    fTable_Be[559, 0] := 2194.37; fTable_Be[559, 1] := 4.04346; fTable_Be[559, 2] := 0.0262870;
    fTable_Be[560, 0] := 2229.86; fTable_Be[560, 1] := 4.04236; fTable_Be[560, 2] := 0.0254127;
    fTable_Be[561, 0] := 2265.93; fTable_Be[561, 1] := 4.04127; fTable_Be[561, 2] := 0.0245675;
    fTable_Be[562, 0] := 2302.57; fTable_Be[562, 1] := 4.04021; fTable_Be[562, 2] := 0.0237503;
    fTable_Be[563, 0] := 2339.82; fTable_Be[563, 1] := 4.03918; fTable_Be[563, 2] := 0.0229604;
    fTable_Be[564, 0] := 2377.66; fTable_Be[564, 1] := 4.03817; fTable_Be[564, 2] := 0.0221967;
    fTable_Be[565, 0] := 2416.12; fTable_Be[565, 1] := 4.03718; fTable_Be[565, 2] := 0.0214584;
    fTable_Be[566, 0] := 2455.20; fTable_Be[566, 1] := 4.03621; fTable_Be[566, 2] := 0.0207447;
    fTable_Be[567, 0] := 2494.91; fTable_Be[567, 1] := 4.03527; fTable_Be[567, 2] := 0.0200547;
    fTable_Be[568, 0] := 2535.26; fTable_Be[568, 1] := 4.03435; fTable_Be[568, 2] := 0.0193877;
    fTable_Be[569, 0] := 2576.27; fTable_Be[569, 1] := 4.03345; fTable_Be[569, 2] := 0.0187429;
    fTable_Be[570, 0] := 2617.94; fTable_Be[570, 1] := 4.03257; fTable_Be[570, 2] := 0.0181195;
    fTable_Be[571, 0] := 2660.28; fTable_Be[571, 1] := 4.03171; fTable_Be[571, 2] := 0.0175168;
    fTable_Be[572, 0] := 2703.31; fTable_Be[572, 1] := 4.03088; fTable_Be[572, 2] := 0.0169342;
    fTable_Be[573, 0] := 2747.03; fTable_Be[573, 1] := 4.03006; fTable_Be[573, 2] := 0.0163709;
    fTable_Be[574, 0] := 2791.46; fTable_Be[574, 1] := 4.02926; fTable_Be[574, 2] := 0.0158264;
    fTable_Be[575, 0] := 2836.61; fTable_Be[575, 1] := 4.02849; fTable_Be[575, 2] := 0.0153000;
    fTable_Be[576, 0] := 2882.49; fTable_Be[576, 1] := 4.02773; fTable_Be[576, 2] := 0.0147911;
    fTable_Be[577, 0] := 2929.11; fTable_Be[577, 1] := 4.02700; fTable_Be[577, 2] := 0.0142992;
    fTable_Be[578, 0] := 2976.49; fTable_Be[578, 1] := 4.02628; fTable_Be[578, 2] := 0.0138236;
    fTable_Be[579, 0] := 3024.63; fTable_Be[579, 1] := 4.02559; fTable_Be[579, 2] := 0.0133638;
    fTable_Be[580, 0] := 3073.55; fTable_Be[580, 1] := 4.02491; fTable_Be[580, 2] := 0.0129072;
    fTable_Be[581, 0] := 3123.26; fTable_Be[581, 1] := 4.02424; fTable_Be[581, 2] := 0.0124663;
    fTable_Be[582, 0] := 3173.78; fTable_Be[582, 1] := 4.02359; fTable_Be[582, 2] := 0.0120403;
    fTable_Be[583, 0] := 3225.11; fTable_Be[583, 1] := 4.02295; fTable_Be[583, 2] := 0.0116290;
    fTable_Be[584, 0] := 3277.28; fTable_Be[584, 1] := 4.02233; fTable_Be[584, 2] := 0.0112317;
    fTable_Be[585, 0] := 3330.29; fTable_Be[585, 1] := 4.02172; fTable_Be[585, 2] := 0.0108480;
    fTable_Be[586, 0] := 3384.15; fTable_Be[586, 1] := 4.02113; fTable_Be[586, 2] := 0.0104774;
    fTable_Be[587, 0] := 3438.89; fTable_Be[587, 1] := 4.02055; fTable_Be[587, 2] := 0.0101194;
    fTable_Be[588, 0] := 3494.51; fTable_Be[588, 1] := 4.01998; fTable_Be[588, 2] := 0.00977365;
    fTable_Be[589, 0] := 3551.03; fTable_Be[589, 1] := 4.01943; fTable_Be[589, 2] := 0.00943974;
    fTable_Be[590, 0] := 3608.46; fTable_Be[590, 1] := 4.01890; fTable_Be[590, 2] := 0.00911724;
    fTable_Be[591, 0] := 3666.83; fTable_Be[591, 1] := 4.01837; fTable_Be[591, 2] := 0.00880575;
    fTable_Be[592, 0] := 3726.13; fTable_Be[592, 1] := 4.01786; fTable_Be[592, 2] := 0.00850491;
    fTable_Be[593, 0] := 3786.40; fTable_Be[593, 1] := 4.01736; fTable_Be[593, 2] := 0.00821432;
    fTable_Be[594, 0] := 3847.64; fTable_Be[594, 1] := 4.01688; fTable_Be[594, 2] := 0.00793369;
    fTable_Be[595, 0] := 3909.88; fTable_Be[595, 1] := 4.01641; fTable_Be[595, 2] := 0.00766264;
    fTable_Be[596, 0] := 3973.12; fTable_Be[596, 1] := 4.01595; fTable_Be[596, 2] := 0.00740085;
    fTable_Be[597, 0] := 4037.38; fTable_Be[597, 1] := 4.01550; fTable_Be[597, 2] := 0.00714801;
    fTable_Be[598, 0] := 4102.68; fTable_Be[598, 1] := 4.01506; fTable_Be[598, 2] := 0.00690380;
    fTable_Be[599, 0] := 4169.04; fTable_Be[599, 1] := 4.01464; fTable_Be[599, 2] := 0.00666401;
    fTable_Be[600, 0] := 4236.47; fTable_Be[600, 1] := 4.01423; fTable_Be[600, 2] := 0.00643256;
    fTable_Be[601, 0] := 4304.99; fTable_Be[601, 1] := 4.01382; fTable_Be[601, 2] := 0.00620915;
    fTable_Be[602, 0] := 4374.62; fTable_Be[602, 1] := 4.01343; fTable_Be[602, 2] := 0.00599350;
    fTable_Be[603, 0] := 4445.37; fTable_Be[603, 1] := 4.01304; fTable_Be[603, 2] := 0.00578535;
    fTable_Be[604, 0] := 4517.27; fTable_Be[604, 1] := 4.01267; fTable_Be[604, 2] := 0.00558442;
    fTable_Be[605, 0] := 4590.34; fTable_Be[605, 1] := 4.01230; fTable_Be[605, 2] := 0.00539045;
    fTable_Be[606, 0] := 4664.58; fTable_Be[606, 1] := 4.01195; fTable_Be[606, 2] := 0.00520323;
    fTable_Be[607, 0] := 4740.03; fTable_Be[607, 1] := 4.01160; fTable_Be[607, 2] := 0.00502252;
    fTable_Be[608, 0] := 4816.70; fTable_Be[608, 1] := 4.01126; fTable_Be[608, 2] := 0.00484809;
    fTable_Be[609, 0] := 4894.60; fTable_Be[609, 1] := 4.01093; fTable_Be[609, 2] := 0.00467971;
    fTable_Be[610, 0] := 4973.77; fTable_Be[610, 1] := 4.01061; fTable_Be[610, 2] := 0.00451716;
    fTable_Be[611, 0] := 5054.21; fTable_Be[611, 1] := 4.01030; fTable_Be[611, 2] := 0.00436028;
    fTable_Be[612, 0] := 5135.96; fTable_Be[612, 1] := 4.01000; fTable_Be[612, 2] := 0.00420884;
    fTable_Be[613, 0] := 5219.03; fTable_Be[613, 1] := 4.00970; fTable_Be[613, 2] := 0.00406267;
    fTable_Be[614, 0] := 5303.45; fTable_Be[614, 1] := 4.00941; fTable_Be[614, 2] := 0.00391977;
    fTable_Be[615, 0] := 5389.23; fTable_Be[615, 1] := 4.00913; fTable_Be[615, 2] := 0.00378191;
    fTable_Be[616, 0] := 5476.39; fTable_Be[616, 1] := 4.00886; fTable_Be[616, 2] := 0.00364888;
    fTable_Be[617, 0] := 5564.97; fTable_Be[617, 1] := 4.00860; fTable_Be[617, 2] := 0.00352054;
    fTable_Be[618, 0] := 5654.98; fTable_Be[618, 1] := 4.00834; fTable_Be[618, 2] := 0.00339671;
    fTable_Be[619, 0] := 5746.44; fTable_Be[619, 1] := 4.00808; fTable_Be[619, 2] := 0.00327724;
    fTable_Be[620, 0] := 5839.39; fTable_Be[620, 1] := 4.00784; fTable_Be[620, 2] := 0.00316197;
    fTable_Be[621, 0] := 5933.83; fTable_Be[621, 1] := 4.00760; fTable_Be[621, 2] := 0.00305075;
    fTable_Be[622, 0] := 6029.81; fTable_Be[622, 1] := 4.00737; fTable_Be[622, 2] := 0.00294344;
    fTable_Be[623, 0] := 6127.33; fTable_Be[623, 1] := 4.00714; fTable_Be[623, 2] := 0.00283992;
    fTable_Be[624, 0] := 6226.44; fTable_Be[624, 1] := 4.00692; fTable_Be[624, 2] := 0.00274003;
    fTable_Be[625, 0] := 6327.15; fTable_Be[625, 1] := 4.00671; fTable_Be[625, 2] := 0.00264365;
    fTable_Be[626, 0] := 6429.48; fTable_Be[626, 1] := 4.00650; fTable_Be[626, 2] := 0.00254975;
    fTable_Be[627, 0] := 6533.48; fTable_Be[627, 1] := 4.00630; fTable_Be[627, 2] := 0.00245918;
    fTable_Be[628, 0] := 6639.15; fTable_Be[628, 1] := 4.00610; fTable_Be[628, 2] := 0.00237183;
    fTable_Be[629, 0] := 6746.53; fTable_Be[629, 1] := 4.00591; fTable_Be[629, 2] := 0.00228759;
    fTable_Be[630, 0] := 6855.65; fTable_Be[630, 1] := 4.00572; fTable_Be[630, 2] := 0.00220633;
    fTable_Be[631, 0] := 6966.54; fTable_Be[631, 1] := 4.00554; fTable_Be[631, 2] := 0.00212796;
    fTable_Be[632, 0] := 7079.21; fTable_Be[632, 1] := 4.00536; fTable_Be[632, 2] := 0.00205238;
    fTable_Be[633, 0] := 7193.71; fTable_Be[633, 1] := 4.00519; fTable_Be[633, 2] := 0.00197947;
    fTable_Be[634, 0] := 7310.07; fTable_Be[634, 1] := 4.00502; fTable_Be[634, 2] := 0.00190916;
    fTable_Be[635, 0] := 7428.30; fTable_Be[635, 1] := 4.00485; fTable_Be[635, 2] := 0.00184135;
    fTable_Be[636, 0] := 7548.45; fTable_Be[636, 1] := 4.00469; fTable_Be[636, 2] := 0.00177595;
    fTable_Be[637, 0] := 7670.54; fTable_Be[637, 1] := 4.00454; fTable_Be[637, 2] := 0.00171287;
    fTable_Be[638, 0] := 7794.60; fTable_Be[638, 1] := 4.00439; fTable_Be[638, 2] := 0.00165202;
    fTable_Be[639, 0] := 7920.68; fTable_Be[639, 1] := 4.00424; fTable_Be[639, 2] := 0.00159334;
    fTable_Be[640, 0] := 8048.79; fTable_Be[640, 1] := 4.00410; fTable_Be[640, 2] := 0.00153675;
    fTable_Be[641, 0] := 8178.97; fTable_Be[641, 1] := 4.00396; fTable_Be[641, 2] := 0.00148216;
    fTable_Be[642, 0] := 8311.26; fTable_Be[642, 1] := 4.00383; fTable_Be[642, 2] := 0.00142952;
    fTable_Be[643, 0] := 8445.68; fTable_Be[643, 1] := 4.00370; fTable_Be[643, 2] := 0.00137819;
    fTable_Be[644, 0] := 8582.29; fTable_Be[644, 1] := 4.00357; fTable_Be[644, 2] := 0.00132870;
    fTable_Be[645, 0] := 8721.10; fTable_Be[645, 1] := 4.00345; fTable_Be[645, 2] := 0.00128099;
    fTable_Be[646, 0] := 8862.16; fTable_Be[646, 1] := 4.00333; fTable_Be[646, 2] := 0.00123499;
    fTable_Be[647, 0] := 9005.49; fTable_Be[647, 1] := 4.00321; fTable_Be[647, 2] := 0.00119064;
    fTable_Be[648, 0] := 9151.15; fTable_Be[648, 1] := 4.00310; fTable_Be[648, 2] := 0.00114789;
    fTable_Be[649, 0] := 9299.16; fTable_Be[649, 1] := 4.00299; fTable_Be[649, 2] := 0.00110667;
    fTable_Be[650, 0] := 9449.57; fTable_Be[650, 1] := 4.00288; fTable_Be[650, 2] := 0.00106693;
    fTable_Be[651, 0] := 9602.41; fTable_Be[651, 1] := 4.00277; fTable_Be[651, 2] := 0.00102862;
    fTable_Be[652, 0] := 9757.72; fTable_Be[652, 1] := 4.00267; fTable_Be[652, 2] := 0.000991686;
    fTable_Be[653, 0] := 9915.54; fTable_Be[653, 1] := 4.00257; fTable_Be[653, 2] := 0.000956077;
    fTable_Be[654, 0] := 10075.9; fTable_Be[654, 1] := 4.00248; fTable_Be[654, 2] := 0.000921746;
    fTable_Be[655, 0] := 10238.9; fTable_Be[655, 1] := 4.00238; fTable_Be[655, 2] := 0.000888646;
    fTable_Be[656, 0] := 10404.5; fTable_Be[656, 1] := 4.00229; fTable_Be[656, 2] := 0.000856737;
    fTable_Be[657, 0] := 10572.8; fTable_Be[657, 1] := 4.00221; fTable_Be[657, 2] := 0.000825973;
    fTable_Be[658, 0] := 10743.8; fTable_Be[658, 1] := 4.00212; fTable_Be[658, 2] := 0.000796314;
    fTable_Be[659, 0] := 10917.6; fTable_Be[659, 1] := 4.00204; fTable_Be[659, 2] := 0.000767721;
    fTable_Be[660, 0] := 11094.1; fTable_Be[660, 1] := 4.00196; fTable_Be[660, 2] := 0.000740154;
    fTable_Be[661, 0] := 11273.6; fTable_Be[661, 1] := 4.00188; fTable_Be[661, 2] := 0.000713574;
    fTable_Be[662, 0] := 11455.9; fTable_Be[662, 1] := 4.00180; fTable_Be[662, 2] := 0.000687952;
    fTable_Be[663, 0] := 11641.2; fTable_Be[663, 1] := 4.00173; fTable_Be[663, 2] := 0.000663249;
    fTable_Be[664, 0] := 11829.5; fTable_Be[664, 1] := 4.00165; fTable_Be[664, 2] := 0.000639433;
    fTable_Be[665, 0] := 12020.8; fTable_Be[665, 1] := 4.00158; fTable_Be[665, 2] := 0.000616473;
    fTable_Be[666, 0] := 12215.3; fTable_Be[666, 1] := 4.00152; fTable_Be[666, 2] := 0.000594337;
    fTable_Be[667, 0] := 12412.8; fTable_Be[667, 1] := 4.00145; fTable_Be[667, 2] := 0.000572994;
    fTable_Be[668, 0] := 12613.6; fTable_Be[668, 1] := 4.00139; fTable_Be[668, 2] := 0.000552174;
    fTable_Be[669, 0] := 12817.6; fTable_Be[669, 1] := 4.00132; fTable_Be[669, 2] := 0.000532111;
    fTable_Be[670, 0] := 13024.9; fTable_Be[670, 1] := 4.00126; fTable_Be[670, 2] := 0.000512776;
    fTable_Be[671, 0] := 13235.6; fTable_Be[671, 1] := 4.00120; fTable_Be[671, 2] := 0.000494145;
    fTable_Be[672, 0] := 13449.7; fTable_Be[672, 1] := 4.00115; fTable_Be[672, 2] := 0.000476188;
    fTable_Be[673, 0] := 13667.2; fTable_Be[673, 1] := 4.00109; fTable_Be[673, 2] := 0.000458886;
    fTable_Be[674, 0] := 13888.3; fTable_Be[674, 1] := 4.00104; fTable_Be[674, 2] := 0.000442212;
    fTable_Be[675, 0] := 14112.9; fTable_Be[675, 1] := 4.00098; fTable_Be[675, 2] := 0.000426144;
    fTable_Be[676, 0] := 14341.2; fTable_Be[676, 1] := 4.00093; fTable_Be[676, 2] := 0.000410660;
    fTable_Be[677, 0] := 14573.1; fTable_Be[677, 1] := 4.00088; fTable_Be[677, 2] := 0.000395739;
    fTable_Be[678, 0] := 14808.8; fTable_Be[678, 1] := 4.00083; fTable_Be[678, 2] := 0.000381358;
    fTable_Be[679, 0] := 15048.3; fTable_Be[679, 1] := 4.00079; fTable_Be[679, 2] := 0.000367502;
    fTable_Be[680, 0] := 15291.7; fTable_Be[680, 1] := 4.00074; fTable_Be[680, 2] := 0.000354148;
    fTable_Be[681, 0] := 15539.1; fTable_Be[681, 1] := 4.00070; fTable_Be[681, 2] := 0.000341280;
    fTable_Be[682, 0] := 15790.4; fTable_Be[682, 1] := 4.00065; fTable_Be[682, 2] := 0.000328880;
    fTable_Be[683, 0] := 16045.8; fTable_Be[683, 1] := 4.00061; fTable_Be[683, 2] := 0.000316929;
    fTable_Be[684, 0] := 16305.3; fTable_Be[684, 1] := 4.00057; fTable_Be[684, 2] := 0.000305413;
    fTable_Be[685, 0] := 16569.1; fTable_Be[685, 1] := 4.00053; fTable_Be[685, 2] := 0.000294207;
    fTable_Be[686, 0] := 16837.0; fTable_Be[686, 1] := 4.00049; fTable_Be[686, 2] := 0.000283413;
    fTable_Be[687, 0] := 17109.4; fTable_Be[687, 1] := 4.00046; fTable_Be[687, 2] := 0.000273015;
    fTable_Be[688, 0] := 17386.1; fTable_Be[688, 1] := 4.00042; fTable_Be[688, 2] := 0.000262998;
    fTable_Be[689, 0] := 17667.3; fTable_Be[689, 1] := 4.00039; fTable_Be[689, 2] := 0.000253348;
    fTable_Be[690, 0] := 17953.1; fTable_Be[690, 1] := 4.00035; fTable_Be[690, 2] := 0.000244052;
    fTable_Be[691, 0] := 18243.4; fTable_Be[691, 1] := 4.00032; fTable_Be[691, 2] := 0.000235098;
    fTable_Be[692, 0] := 18538.5; fTable_Be[692, 1] := 4.00029; fTable_Be[692, 2] := 0.000226472;
    fTable_Be[693, 0] := 18838.4; fTable_Be[693, 1] := 4.00026; fTable_Be[693, 2] := 0.000218163;
    fTable_Be[694, 0] := 19143.0; fTable_Be[694, 1] := 4.00023; fTable_Be[694, 2] := 0.000210159;
    fTable_Be[695, 0] := 19452.7; fTable_Be[695, 1] := 4.00020; fTable_Be[695, 2] := 0.000202447;
    fTable_Be[696, 0] := 19767.3; fTable_Be[696, 1] := 4.00017; fTable_Be[696, 2] := 0.000195019;
    fTable_Be[697, 0] := 20087.0; fTable_Be[697, 1] := 4.00014; fTable_Be[697, 2] := 0.000187864;
    fTable_Be[698, 0] := 20411.9; fTable_Be[698, 1] := 4.00011; fTable_Be[698, 2] := 0.000180971;
    fTable_Be[699, 0] := 20742.1; fTable_Be[699, 1] := 4.00009; fTable_Be[699, 2] := 0.000174332;
    fTable_Be[700, 0] := 21077.5; fTable_Be[700, 1] := 4.00006; fTable_Be[700, 2] := 0.000167935;
    fTable_Be[701, 0] := 21418.5; fTable_Be[701, 1] := 4.00004; fTable_Be[701, 2] := 0.000161773;
    fTable_Be[702, 0] := 21764.9; fTable_Be[702, 1] := 4.00001; fTable_Be[702, 2] := 0.000155838;
    fTable_Be[703, 0] := 22116.9; fTable_Be[703, 1] := 3.99999; fTable_Be[703, 2] := 0.000150120;
    fTable_Be[704, 0] := 22474.6; fTable_Be[704, 1] := 3.99997; fTable_Be[704, 2] := 0.000144612;
    fTable_Be[705, 0] := 22838.1; fTable_Be[705, 1] := 3.99995; fTable_Be[705, 2] := 0.000139307;
    fTable_Be[706, 0] := 23207.5; fTable_Be[706, 1] := 3.99992; fTable_Be[706, 2] := 0.000134195;
    fTable_Be[707, 0] := 23582.9; fTable_Be[707, 1] := 3.99990; fTable_Be[707, 2] := 0.000129271;
    fTable_Be[708, 0] := 23964.3; fTable_Be[708, 1] := 3.99988; fTable_Be[708, 2] := 0.000124528;
    fTable_Be[709, 0] := 24351.9; fTable_Be[709, 1] := 3.99986; fTable_Be[709, 2] := 0.000119959;
    fTable_Be[710, 0] := 24745.8; fTable_Be[710, 1] := 3.99985; fTable_Be[710, 2] := 0.000115558;
    fTable_Be[711, 0] := 25146.1; fTable_Be[711, 1] := 3.99983; fTable_Be[711, 2] := 0.000111318;
    fTable_Be[712, 0] := 25552.8; fTable_Be[712, 1] := 3.99981; fTable_Be[712, 2] := 0.000107234;
    fTable_Be[713, 0] := 25966.1; fTable_Be[713, 1] := 3.99979; fTable_Be[713, 2] := 0.000103299;
    fTable_Be[714, 0] := 26386.0; fTable_Be[714, 1] := 3.99978; fTable_Be[714, 2] := 0.0000995092;
    fTable_Be[715, 0] := 26812.8; fTable_Be[715, 1] := 3.99976; fTable_Be[715, 2] := 0.0000958583;
    fTable_Be[716, 0] := 27246.5; fTable_Be[716, 1] := 3.99974; fTable_Be[716, 2] := 0.0000923412;
    fTable_Be[717, 0] := 27687.2; fTable_Be[717, 1] := 3.99973; fTable_Be[717, 2] := 0.0000889532;
    fTable_Be[718, 0] := 28135.0; fTable_Be[718, 1] := 3.99971; fTable_Be[718, 2] := 0.0000856893;
    fTable_Be[719, 0] := 28590.1; fTable_Be[719, 1] := 3.99970; fTable_Be[719, 2] := 0.0000825453;
    fTable_Be[720, 0] := 29052.5; fTable_Be[720, 1] := 3.99969; fTable_Be[720, 2] := 0.0000795168;
    fTable_Be[721, 0] := 29522.4; fTable_Be[721, 1] := 3.99967; fTable_Be[721, 2] := 0.0000765993;
    fTable_Be[722, 0] := 29999.9; fTable_Be[722, 1] := 3.99966; fTable_Be[722, 2] := 0.0000737888;
    fTable_Be[723, 0] := 30000.0; fTable_Be[723, 1] := 3.99966; fTable_Be[723, 2] := 0.0000737882;

    (* Table initialization: fTable_Si *)
    fTable_Si[0, 0] := 10.0000; fTable_Si[0, 1] := -9999; fTable_Si[0, 2] := 3.94851;
    fTable_Si[1, 0] := 10.1617; fTable_Si[1, 1] := -9999; fTable_Si[1, 2] := 3.95531;
    fTable_Si[2, 0] := 10.3261; fTable_Si[2, 1] := -9999; fTable_Si[2, 2] := 3.96212;
    fTable_Si[3, 0] := 10.4931; fTable_Si[3, 1] := -9999; fTable_Si[3, 2] := 3.96894;
    fTable_Si[4, 0] := 10.6628; fTable_Si[4, 1] := -9999; fTable_Si[4, 2] := 3.97577;
    fTable_Si[5, 0] := 10.8353; fTable_Si[5, 1] := -9999; fTable_Si[5, 2] := 3.98262;
    fTable_Si[6, 0] := 11.0105; fTable_Si[6, 1] := -9999; fTable_Si[6, 2] := 3.98948;
    fTable_Si[7, 0] := 11.1886; fTable_Si[7, 1] := -9999; fTable_Si[7, 2] := 3.99635;
    fTable_Si[8, 0] := 11.3696; fTable_Si[8, 1] := -9999; fTable_Si[8, 2] := 4.00322;
    fTable_Si[9, 0] := 11.5535; fTable_Si[9, 1] := -9999; fTable_Si[9, 2] := 4.01012;
    fTable_Si[10, 0] := 11.7404; fTable_Si[10, 1] := -9999; fTable_Si[10, 2] := 4.01702;
    fTable_Si[11, 0] := 11.9303; fTable_Si[11, 1] := -9999; fTable_Si[11, 2] := 4.02394;
    fTable_Si[12, 0] := 12.1232; fTable_Si[12, 1] := -9999; fTable_Si[12, 2] := 4.00019;
    fTable_Si[13, 0] := 12.3193; fTable_Si[13, 1] := -9999; fTable_Si[13, 2] := 3.95930;
    fTable_Si[14, 0] := 12.5186; fTable_Si[14, 1] := -9999; fTable_Si[14, 2] := 3.91883;
    fTable_Si[15, 0] := 12.7210; fTable_Si[15, 1] := -9999; fTable_Si[15, 2] := 3.87876;
    fTable_Si[16, 0] := 12.9268; fTable_Si[16, 1] := -9999; fTable_Si[16, 2] := 3.83911;
    fTable_Si[17, 0] := 13.1359; fTable_Si[17, 1] := -9999; fTable_Si[17, 2] := 3.79987;
    fTable_Si[18, 0] := 13.3483; fTable_Si[18, 1] := -9999; fTable_Si[18, 2] := 3.76102;
    fTable_Si[19, 0] := 13.5642; fTable_Si[19, 1] := -9999; fTable_Si[19, 2] := 3.72257;
    fTable_Si[20, 0] := 13.7836; fTable_Si[20, 1] := -9999; fTable_Si[20, 2] := 3.68452;
    fTable_Si[21, 0] := 14.0066; fTable_Si[21, 1] := -9999; fTable_Si[21, 2] := 3.64513;
    fTable_Si[22, 0] := 14.2331; fTable_Si[22, 1] := -9999; fTable_Si[22, 2] := 3.55020;
    fTable_Si[23, 0] := 14.4633; fTable_Si[23, 1] := -9999; fTable_Si[23, 2] := 3.45774;
    fTable_Si[24, 0] := 14.6972; fTable_Si[24, 1] := -9999; fTable_Si[24, 2] := 3.36769;
    fTable_Si[25, 0] := 14.9350; fTable_Si[25, 1] := -9999; fTable_Si[25, 2] := 3.27998;
    fTable_Si[26, 0] := 15.1765; fTable_Si[26, 1] := -9999; fTable_Si[26, 2] := 3.19455;
    fTable_Si[27, 0] := 15.4220; fTable_Si[27, 1] := -9999; fTable_Si[27, 2] := 3.11136;
    fTable_Si[28, 0] := 15.6714; fTable_Si[28, 1] := -9999; fTable_Si[28, 2] := 3.03032;
    fTable_Si[29, 0] := 15.9249; fTable_Si[29, 1] := -9999; fTable_Si[29, 2] := 2.95140;
    fTable_Si[30, 0] := 16.1825; fTable_Si[30, 1] := -9999; fTable_Si[30, 2] := 2.83114;
    fTable_Si[31, 0] := 16.4442; fTable_Si[31, 1] := -9999; fTable_Si[31, 2] := 2.69869;
    fTable_Si[32, 0] := 16.7102; fTable_Si[32, 1] := -9999; fTable_Si[32, 2] := 2.57244;
    fTable_Si[33, 0] := 16.9805; fTable_Si[33, 1] := -9999; fTable_Si[33, 2] := 2.45210;
    fTable_Si[34, 0] := 17.2551; fTable_Si[34, 1] := -9999; fTable_Si[34, 2] := 2.33738;
    fTable_Si[35, 0] := 17.5342; fTable_Si[35, 1] := -9999; fTable_Si[35, 2] := 2.22803;
    fTable_Si[36, 0] := 17.8178; fTable_Si[36, 1] := -9999; fTable_Si[36, 2] := 2.12380;
    fTable_Si[37, 0] := 18.1060; fTable_Si[37, 1] := -9999; fTable_Si[37, 2] := 1.97554;
    fTable_Si[38, 0] := 18.3988; fTable_Si[38, 1] := -9999; fTable_Si[38, 2] := 1.76138;
    fTable_Si[39, 0] := 18.6964; fTable_Si[39, 1] := -9999; fTable_Si[39, 2] := 1.57043;
    fTable_Si[40, 0] := 18.9988; fTable_Si[40, 1] := -9999; fTable_Si[40, 2] := 1.40019;
    fTable_Si[41, 0] := 19.3061; fTable_Si[41, 1] := -9999; fTable_Si[41, 2] := 1.24840;
    fTable_Si[42, 0] := 19.6184; fTable_Si[42, 1] := -9999; fTable_Si[42, 2] := 1.11306;
    fTable_Si[43, 0] := 19.9357; fTable_Si[43, 1] := -9999; fTable_Si[43, 2] := 0.992396;
    fTable_Si[44, 0] := 20.2581; fTable_Si[44, 1] := -9999; fTable_Si[44, 2] := 0.862336;
    fTable_Si[45, 0] := 20.5858; fTable_Si[45, 1] := -9999; fTable_Si[45, 2] := 0.753564;
    fTable_Si[46, 0] := 20.9187; fTable_Si[46, 1] := -9999; fTable_Si[46, 2] := 0.698871;
    fTable_Si[47, 0] := 21.2571; fTable_Si[47, 1] := -9999; fTable_Si[47, 2] := 0.648148;
    fTable_Si[48, 0] := 21.6009; fTable_Si[48, 1] := -9999; fTable_Si[48, 2] := 0.602543;
    fTable_Si[49, 0] := 21.9503; fTable_Si[49, 1] := -9999; fTable_Si[49, 2] := 0.561516;
    fTable_Si[50, 0] := 22.3053; fTable_Si[50, 1] := -9999; fTable_Si[50, 2] := 0.523281;
    fTable_Si[51, 0] := 22.6661; fTable_Si[51, 1] := -9999; fTable_Si[51, 2] := 0.496895;
    fTable_Si[52, 0] := 23.0327; fTable_Si[52, 1] := -9999; fTable_Si[52, 2] := 0.478071;
    fTable_Si[53, 0] := 23.4052; fTable_Si[53, 1] := -9999; fTable_Si[53, 2] := 0.459962;
    fTable_Si[54, 0] := 23.7838; fTable_Si[54, 1] := -9999; fTable_Si[54, 2] := 0.442538;
    fTable_Si[55, 0] := 24.1685; fTable_Si[55, 1] := -9999; fTable_Si[55, 2] := 0.425774;
    fTable_Si[56, 0] := 24.5594; fTable_Si[56, 1] := -9999; fTable_Si[56, 2] := 0.413096;
    fTable_Si[57, 0] := 24.9566; fTable_Si[57, 1] := -9999; fTable_Si[57, 2] := 0.403041;
    fTable_Si[58, 0] := 25.3602; fTable_Si[58, 1] := -9999; fTable_Si[58, 2] := 0.393231;
    fTable_Si[59, 0] := 25.7704; fTable_Si[59, 1] := -9999; fTable_Si[59, 2] := 0.383660;
    fTable_Si[60, 0] := 26.1872; fTable_Si[60, 1] := -9999; fTable_Si[60, 2] := 0.374321;
    fTable_Si[61, 0] := 26.6108; fTable_Si[61, 1] := -9999; fTable_Si[61, 2] := 0.365210;
    fTable_Si[62, 0] := 27.0412; fTable_Si[62, 1] := -9999; fTable_Si[62, 2] := 0.366288;
    fTable_Si[63, 0] := 27.4786; fTable_Si[63, 1] := -9999; fTable_Si[63, 2] := 0.367374;
    fTable_Si[64, 0] := 27.9230; fTable_Si[64, 1] := -9999; fTable_Si[64, 2] := 0.368463;
    fTable_Si[65, 0] := 28.3747; fTable_Si[65, 1] := -9999; fTable_Si[65, 2] := 0.369555;
    fTable_Si[66, 0] := 28.8336; fTable_Si[66, 1] := -9999; fTable_Si[66, 2] := 0.370650;
    fTable_Si[67, 0] := 29.3000; fTable_Si[67, 1] := 3.83380; fTable_Si[67, 2] := 0.371749;
    fTable_Si[68, 0] := 29.7739; fTable_Si[68, 1] := 3.80691; fTable_Si[68, 2] := 0.372851;
    fTable_Si[69, 0] := 30.2554; fTable_Si[69, 1] := 3.78097; fTable_Si[69, 2] := 0.373956;
    fTable_Si[70, 0] := 30.7448; fTable_Si[70, 1] := 3.75582; fTable_Si[70, 2] := 0.375064;
    fTable_Si[71, 0] := 31.2421; fTable_Si[71, 1] := 3.73048; fTable_Si[71, 2] := 0.376176;
    fTable_Si[72, 0] := 31.7474; fTable_Si[72, 1] := 3.70550; fTable_Si[72, 2] := 0.378088;
    fTable_Si[73, 0] := 32.2609; fTable_Si[73, 1] := 3.68147; fTable_Si[73, 2] := 0.381996;
    fTable_Si[74, 0] := 32.7827; fTable_Si[74, 1] := 3.65905; fTable_Si[74, 2] := 0.385945;
    fTable_Si[75, 0] := 33.3129; fTable_Si[75, 1] := 3.63764; fTable_Si[75, 2] := 0.389935;
    fTable_Si[76, 0] := 33.8517; fTable_Si[76, 1] := 3.61703; fTable_Si[76, 2] := 0.393965;
    fTable_Si[77, 0] := 34.3992; fTable_Si[77, 1] := 3.59711; fTable_Si[77, 2] := 0.398038;
    fTable_Si[78, 0] := 34.9556; fTable_Si[78, 1] := 3.57779; fTable_Si[78, 2] := 0.402152;
    fTable_Si[79, 0] := 35.5210; fTable_Si[79, 1] := 3.55900; fTable_Si[79, 2] := 0.406309;
    fTable_Si[80, 0] := 36.0955; fTable_Si[80, 1] := 3.54071; fTable_Si[80, 2] := 0.410509;
    fTable_Si[81, 0] := 36.6793; fTable_Si[81, 1] := 3.52286; fTable_Si[81, 2] := 0.414753;
    fTable_Si[82, 0] := 37.2726; fTable_Si[82, 1] := 3.50545; fTable_Si[82, 2] := 0.419040;
    fTable_Si[83, 0] := 37.8754; fTable_Si[83, 1] := 3.48848; fTable_Si[83, 2] := 0.423372;
    fTable_Si[84, 0] := 38.4880; fTable_Si[84, 1] := 3.47200; fTable_Si[84, 2] := 0.427748;
    fTable_Si[85, 0] := 39.1106; fTable_Si[85, 1] := 3.45628; fTable_Si[85, 2] := 0.432170;
    fTable_Si[86, 0] := 39.7431; fTable_Si[86, 1] := 3.44176; fTable_Si[86, 2] := 0.435537;
    fTable_Si[87, 0] := 40.3860; fTable_Si[87, 1] := 3.42689; fTable_Si[87, 2] := 0.437136;
    fTable_Si[88, 0] := 41.0392; fTable_Si[88, 1] := 3.41050; fTable_Si[88, 2] := 0.438741;
    fTable_Si[89, 0] := 41.7029; fTable_Si[89, 1] := 3.39378; fTable_Si[89, 2] := 0.440351;
    fTable_Si[90, 0] := 42.3774; fTable_Si[90, 1] := 3.37667; fTable_Si[90, 2] := 0.441968;
    fTable_Si[91, 0] := 43.0629; fTable_Si[91, 1] := 3.35917; fTable_Si[91, 2] := 0.443590;
    fTable_Si[92, 0] := 43.7594; fTable_Si[92, 1] := 3.34130; fTable_Si[92, 2] := 0.445218;
    fTable_Si[93, 0] := 44.4671; fTable_Si[93, 1] := 3.32304; fTable_Si[93, 2] := 0.446852;
    fTable_Si[94, 0] := 45.1864; fTable_Si[94, 1] := 3.30440; fTable_Si[94, 2] := 0.448493;
    fTable_Si[95, 0] := 45.9172; fTable_Si[95, 1] := 3.28549; fTable_Si[95, 2] := 0.450139;
    fTable_Si[96, 0] := 46.6599; fTable_Si[96, 1] := 3.26615; fTable_Si[96, 2] := 0.451198;
    fTable_Si[97, 0] := 47.4146; fTable_Si[97, 1] := 3.24599; fTable_Si[97, 2] := 0.451979;
    fTable_Si[98, 0] := 48.1815; fTable_Si[98, 1] := 3.22476; fTable_Si[98, 2] := 0.452762;
    fTable_Si[99, 0] := 48.9608; fTable_Si[99, 1] := 3.20267; fTable_Si[99, 2] := 0.453547;
    fTable_Si[100, 0] := 49.7527; fTable_Si[100, 1] := 3.17964; fTable_Si[100, 2] := 0.454332;
    fTable_Si[101, 0] := 50.5574; fTable_Si[101, 1] := 3.15558; fTable_Si[101, 2] := 0.455119;
    fTable_Si[102, 0] := 51.3751; fTable_Si[102, 1] := 3.13042; fTable_Si[102, 2] := 0.455908;
    fTable_Si[103, 0] := 52.2061; fTable_Si[103, 1] := 3.10325; fTable_Si[103, 2] := 0.456698;
    fTable_Si[104, 0] := 53.0505; fTable_Si[104, 1] := 3.07444; fTable_Si[104, 2] := 0.458301;
    fTable_Si[105, 0] := 53.9085; fTable_Si[105, 1] := 3.04507; fTable_Si[105, 2] := 0.461948;
    fTable_Si[106, 0] := 54.7804; fTable_Si[106, 1] := 3.01545; fTable_Si[106, 2] := 0.465624;
    fTable_Si[107, 0] := 55.6665; fTable_Si[107, 1] := 2.98498; fTable_Si[107, 2] := 0.469328;
    fTable_Si[108, 0] := 56.5668; fTable_Si[108, 1] := 2.95338; fTable_Si[108, 2] := 0.473062;
    fTable_Si[109, 0] := 57.4817; fTable_Si[109, 1] := 2.92040; fTable_Si[109, 2] := 0.476826;
    fTable_Si[110, 0] := 58.4115; fTable_Si[110, 1] := 2.88519; fTable_Si[110, 2] := 0.480620;
    fTable_Si[111, 0] := 59.3562; fTable_Si[111, 1] := 2.84598; fTable_Si[111, 2] := 0.484444;
    fTable_Si[112, 0] := 60.3163; fTable_Si[112, 1] := 2.80606; fTable_Si[112, 2] := 0.494947;
    fTable_Si[113, 0] := 61.2918; fTable_Si[113, 1] := 2.76788; fTable_Si[113, 2] := 0.506504;
    fTable_Si[114, 0] := 62.2832; fTable_Si[114, 1] := 2.73042; fTable_Si[114, 2] := 0.518332;
    fTable_Si[115, 0] := 63.2906; fTable_Si[115, 1] := 2.69333; fTable_Si[115, 2] := 0.530436;
    fTable_Si[116, 0] := 64.3142; fTable_Si[116, 1] := 2.65696; fTable_Si[116, 2] := 0.542822;
    fTable_Si[117, 0] := 65.3545; fTable_Si[117, 1] := 2.62418; fTable_Si[117, 2] := 0.554884;
    fTable_Si[118, 0] := 66.4115; fTable_Si[118, 1] := 2.58874; fTable_Si[118, 2] := 0.558968;
    fTable_Si[119, 0] := 67.4857; fTable_Si[119, 1] := 2.54971; fTable_Si[119, 2] := 0.563081;
    fTable_Si[120, 0] := 68.5772; fTable_Si[120, 1] := 2.50917; fTable_Si[120, 2] := 0.567224;
    fTable_Si[121, 0] := 69.6864; fTable_Si[121, 1] := 2.46935; fTable_Si[121, 2] := 0.571398;
    fTable_Si[122, 0] := 70.8135; fTable_Si[122, 1] := 2.43129; fTable_Si[122, 2] := 0.566814;
    fTable_Si[123, 0] := 71.9588; fTable_Si[123, 1] := 2.38275; fTable_Si[123, 2] := 0.552979;
    fTable_Si[124, 0] := 73.1227; fTable_Si[124, 1] := 2.32504; fTable_Si[124, 2] := 0.539483;
    fTable_Si[125, 0] := 74.3054; fTable_Si[125, 1] := 2.26322; fTable_Si[125, 2] := 0.526316;
    fTable_Si[126, 0] := 75.5072; fTable_Si[126, 1] := 2.19828; fTable_Si[126, 2] := 0.504782;
    fTable_Si[127, 0] := 76.7285; fTable_Si[127, 1] := 2.11635; fTable_Si[127, 2] := 0.477417;
    fTable_Si[128, 0] := 77.9695; fTable_Si[128, 1] := 2.01618; fTable_Si[128, 2] := 0.451535;
    fTable_Si[129, 0] := 79.2306; fTable_Si[129, 1] := 1.90170; fTable_Si[129, 2] := 0.427364;
    fTable_Si[130, 0] := 80.5121; fTable_Si[130, 1] := 1.77437; fTable_Si[130, 2] := 0.422623;
    fTable_Si[131, 0] := 81.8143; fTable_Si[131, 1] := 1.64458; fTable_Si[131, 2] := 0.417936;
    fTable_Si[132, 0] := 83.1376; fTable_Si[132, 1] := 1.50518; fTable_Si[132, 2] := 0.413300;
    fTable_Si[133, 0] := 84.4823; fTable_Si[133, 1] := 1.34727; fTable_Si[133, 2] := 0.409326;
    fTable_Si[134, 0] := 85.8487; fTable_Si[134, 1] := 1.17621; fTable_Si[134, 2] := 0.415946;
    fTable_Si[135, 0] := 87.2373; fTable_Si[135, 1] := 0.995339; fTable_Si[135, 2] := 0.422674;
    fTable_Si[136, 0] := 88.6483; fTable_Si[136, 1] := 0.794497; fTable_Si[136, 2] := 0.429510;
    fTable_Si[137, 0] := 90.0821; fTable_Si[137, 1] := 0.568059; fTable_Si[137, 2] := 0.436457;
    fTable_Si[138, 0] := 91.5391; fTable_Si[138, 1] := 0.306962; fTable_Si[138, 2] := 0.444926;
    fTable_Si[139, 0] := 93.0197; fTable_Si[139, 1] := 0.00161588; fTable_Si[139, 2] := 0.456528;
    fTable_Si[140, 0] := 94.5242; fTable_Si[140, 1] := -0.366911; fTable_Si[140, 2] := 0.468434;
    fTable_Si[141, 0] := 96.0530; fTable_Si[141, 1] := -0.841388; fTable_Si[141, 2] := 0.480650;
    fTable_Si[142, 0] := 97.6066; fTable_Si[142, 1] := -1.52605; fTable_Si[142, 2] := 0.495035;
    fTable_Si[143, 0] := 99.1853; fTable_Si[143, 1] := -2.88115; fTable_Si[143, 2] := 0.517644;
    fTable_Si[144, 0] := 99.5000; fTable_Si[144, 1] := -3.50392; fTable_Si[144, 2] := 0.522228;
    fTable_Si[145, 0] := 99.5240; fTable_Si[145, 1] := -3.56793; fTable_Si[145, 2] := 0.517644;
    fTable_Si[146, 0] := 99.5490; fTable_Si[146, 1] := -3.65086; fTable_Si[146, 2] := 0.517841;
    fTable_Si[147, 0] := 99.5760; fTable_Si[147, 1] := -3.74861; fTable_Si[147, 2] := 0.521284;
    fTable_Si[148, 0] := 99.6010; fTable_Si[148, 1] := -3.84977; fTable_Si[148, 2] := 0.535297;
    fTable_Si[149, 0] := 99.6260; fTable_Si[149, 1] := -3.95788; fTable_Si[149, 2] := 0.552022;
    fTable_Si[150, 0] := 99.6490; fTable_Si[150, 1] := -4.07048; fTable_Si[150, 2] := 0.581748;
    fTable_Si[151, 0] := 99.6760; fTable_Si[151, 1] := -4.21370; fTable_Si[151, 2] := 0.630001;
    fTable_Si[152, 0] := 99.6990; fTable_Si[152, 1] := -4.33738; fTable_Si[152, 2] := 0.708784;
    fTable_Si[153, 0] := 99.7260; fTable_Si[153, 1] := -4.47439; fTable_Si[153, 2] := 0.813415;
    fTable_Si[154, 0] := 99.7490; fTable_Si[154, 1] := -4.57087; fTable_Si[154, 2] := 0.941569;
    fTable_Si[155, 0] := 99.7750; fTable_Si[155, 1] := -4.65499; fTable_Si[155, 2] := 1.07721;
    fTable_Si[156, 0] := 99.8260; fTable_Si[156, 1] := -4.76959; fTable_Si[156, 2] := 1.37513;
    fTable_Si[157, 0] := 99.8510; fTable_Si[157, 1] := -4.79109; fTable_Si[157, 2] := 1.52203;
    fTable_Si[158, 0] := 99.8750; fTable_Si[158, 1] := -4.78699; fTable_Si[158, 2] := 1.65993;
    fTable_Si[159, 0] := 99.8990; fTable_Si[159, 1] := -4.76674; fTable_Si[159, 2] := 1.77995;
    fTable_Si[160, 0] := 99.9260; fTable_Si[160, 1] := -4.73984; fTable_Si[160, 2] := 1.87968;
    fTable_Si[161, 0] := 99.9510; fTable_Si[161, 1] := -4.72571; fTable_Si[161, 2] := 1.97448;
    fTable_Si[162, 0] := 99.9740; fTable_Si[162, 1] := -4.69897; fTable_Si[162, 2] := 2.05815;
    fTable_Si[163, 0] := 100.000; fTable_Si[163, 1] := -4.67405; fTable_Si[163, 2] := 2.13311;
    fTable_Si[164, 0] := 100.030; fTable_Si[164, 1] := -4.65490; fTable_Si[164, 2] := 2.20171;
    fTable_Si[165, 0] := 100.120; fTable_Si[165, 1] := -4.60024; fTable_Si[165, 2] := 2.41667;
    fTable_Si[166, 0] := 100.180; fTable_Si[166, 1] := -4.60059; fTable_Si[166, 2] := 2.49729;
    fTable_Si[167, 0] := 100.220; fTable_Si[167, 1] := -4.62085; fTable_Si[167, 2] := 2.58505;
    fTable_Si[168, 0] := 100.250; fTable_Si[168, 1] := -4.64510; fTable_Si[168, 2] := 2.62089;
    fTable_Si[169, 0] := 100.280; fTable_Si[169, 1] := -4.70275; fTable_Si[169, 2] := 2.67241;
    fTable_Si[170, 0] := 100.300; fTable_Si[170, 1] := -4.73916; fTable_Si[170, 2] := 2.73072;
    fTable_Si[171, 0] := 100.350; fTable_Si[171, 1] := -4.82406; fTable_Si[171, 2] := 2.91360;
    fTable_Si[172, 0] := 100.380; fTable_Si[172, 1] := -4.87754; fTable_Si[172, 2] := 3.01959;
    fTable_Si[173, 0] := 100.450; fTable_Si[173, 1] := -4.89461; fTable_Si[173, 2] := 3.39622;
    fTable_Si[174, 0] := 100.480; fTable_Si[174, 1] := -4.89177; fTable_Si[174, 2] := 3.52655;
    fTable_Si[175, 0] := 100.500; fTable_Si[175, 1] := -4.87133; fTable_Si[175, 2] := 3.64732;
    fTable_Si[176, 0] := 100.550; fTable_Si[176, 1] := -4.80557; fTable_Si[176, 2] := 3.86847;
    fTable_Si[177, 0] := 100.600; fTable_Si[177, 1] := -4.71048; fTable_Si[177, 2] := 4.10668;
    fTable_Si[178, 0] := 100.620; fTable_Si[178, 1] := -4.63514; fTable_Si[178, 2] := 4.23678;
    fTable_Si[179, 0] := 100.680; fTable_Si[179, 1] := -4.54337; fTable_Si[179, 2] := 4.36464;
    fTable_Si[180, 0] := 100.700; fTable_Si[180, 1] := -4.48607; fTable_Si[180, 2] := 4.49509;
    fTable_Si[181, 0] := 100.750; fTable_Si[181, 1] := -4.33702; fTable_Si[181, 2] := 4.75764;
    fTable_Si[182, 0] := 100.770; fTable_Si[182, 1] := -4.23325; fTable_Si[182, 2] := 4.85961;
    fTable_Si[183, 0] := 100.800; fTable_Si[183, 1] := -4.07337; fTable_Si[183, 2] := 4.94637;
    fTable_Si[184, 0] := 100.850; fTable_Si[184, 1] := -3.81798; fTable_Si[184, 2] := 5.07430;
    fTable_Si[185, 0] := 100.900; fTable_Si[185, 1] := -3.56548; fTable_Si[185, 2] := 5.12335;
    fTable_Si[186, 0] := 101.000; fTable_Si[186, 1] := -3.15785; fTable_Si[186, 2] := 5.13032;
    fTable_Si[187, 0] := 101.020; fTable_Si[187, 1] := -3.08861; fTable_Si[187, 2] := 5.12048;
    fTable_Si[188, 0] := 101.250; fTable_Si[188, 1] := -2.52100; fTable_Si[188, 2] := 5.15904;
    fTable_Si[189, 0] := 101.320; fTable_Si[189, 1] := -2.30405; fTable_Si[189, 2] := 5.19959;
    fTable_Si[190, 0] := 101.380; fTable_Si[190, 1] := -2.08534; fTable_Si[190, 2] := 5.20146;
    fTable_Si[191, 0] := 101.400; fTable_Si[191, 1] := -2.00971; fTable_Si[191, 2] := 5.18989;
    fTable_Si[192, 0] := 101.450; fTable_Si[192, 1] := -1.81270; fTable_Si[192, 2] := 5.13442;
    fTable_Si[193, 0] := 101.500; fTable_Si[193, 1] := -1.65152; fTable_Si[193, 2] := 5.02977;
    fTable_Si[194, 0] := 101.600; fTable_Si[194, 1] := -1.41105; fTable_Si[194, 2] := 4.78618;
    fTable_Si[195, 0] := 101.630; fTable_Si[195, 1] := -1.36359; fTable_Si[195, 2] := 4.72648;
    fTable_Si[196, 0] := 101.650; fTable_Si[196, 1] := -1.35292; fTable_Si[196, 2] := 4.65861;
    fTable_Si[197, 0] := 101.750; fTable_Si[197, 1] := -1.25455; fTable_Si[197, 2] := 4.44125;
    fTable_Si[198, 0] := 101.820; fTable_Si[198, 1] := -1.21389; fTable_Si[198, 2] := 4.30165;
    fTable_Si[199, 0] := 101.880; fTable_Si[199, 1] := -1.19458; fTable_Si[199, 2] := 4.18620;
    fTable_Si[200, 0] := 101.900; fTable_Si[200, 1] := -1.20985; fTable_Si[200, 2] := 4.13288;
    fTable_Si[201, 0] := 101.950; fTable_Si[201, 1] := -1.20581; fTable_Si[201, 2] := 4.08850;
    fTable_Si[202, 0] := 102.000; fTable_Si[202, 1] := -1.19801; fTable_Si[202, 2] := 3.97606;
    fTable_Si[203, 0] := 102.030; fTable_Si[203, 1] := -1.22710; fTable_Si[203, 2] := 3.93010;
    fTable_Si[204, 0] := 102.050; fTable_Si[204, 1] := -1.24904; fTable_Si[204, 2] := 3.89784;
    fTable_Si[205, 0] := 102.100; fTable_Si[205, 1] := -1.28103; fTable_Si[205, 2] := 3.86731;
    fTable_Si[206, 0] := 102.150; fTable_Si[206, 1] := -1.30990; fTable_Si[206, 2] := 3.80579;
    fTable_Si[207, 0] := 102.180; fTable_Si[207, 1] := -1.33991; fTable_Si[207, 2] := 3.78427;
    fTable_Si[208, 0] := 102.250; fTable_Si[208, 1] := -1.39700; fTable_Si[208, 2] := 3.76802;
    fTable_Si[209, 0] := 102.300; fTable_Si[209, 1] := -1.42608; fTable_Si[209, 2] := 3.74849;
    fTable_Si[210, 0] := 102.350; fTable_Si[210, 1] := -1.46728; fTable_Si[210, 2] := 3.74261;
    fTable_Si[211, 0] := 102.400; fTable_Si[211, 1] := -1.50309; fTable_Si[211, 2] := 3.76084;
    fTable_Si[212, 0] := 102.450; fTable_Si[212, 1] := -1.52538; fTable_Si[212, 2] := 3.79386;
    fTable_Si[213, 0] := 102.530; fTable_Si[213, 1] := -1.50608; fTable_Si[213, 2] := 3.87484;
    fTable_Si[214, 0] := 102.550; fTable_Si[214, 1] := -1.48153; fTable_Si[214, 2] := 3.89373;
    fTable_Si[215, 0] := 102.600; fTable_Si[215, 1] := -1.42009; fTable_Si[215, 2] := 3.90179;
    fTable_Si[216, 0] := 102.650; fTable_Si[216, 1] := -1.36279; fTable_Si[216, 2] := 3.88239;
    fTable_Si[217, 0] := 102.700; fTable_Si[217, 1] := -1.31820; fTable_Si[217, 2] := 3.83958;
    fTable_Si[218, 0] := 102.780; fTable_Si[218, 1] := -1.29202; fTable_Si[218, 2] := 3.76416;
    fTable_Si[219, 0] := 102.880; fTable_Si[219, 1] := -1.29963; fTable_Si[219, 2] := 3.67993;
    fTable_Si[220, 0] := 102.950; fTable_Si[220, 1] := -1.32951; fTable_Si[220, 2] := 3.64539;
    fTable_Si[221, 0] := 103.000; fTable_Si[221, 1] := -1.34633; fTable_Si[221, 2] := 3.63286;
    fTable_Si[222, 0] := 103.120; fTable_Si[222, 1] := -1.36198; fTable_Si[222, 2] := 3.65919;
    fTable_Si[223, 0] := 103.200; fTable_Si[223, 1] := -1.32264; fTable_Si[223, 2] := 3.65521;
    fTable_Si[224, 0] := 103.280; fTable_Si[224, 1] := -1.27117; fTable_Si[224, 2] := 3.62578;
    fTable_Si[225, 0] := 103.320; fTable_Si[225, 1] := -1.25882; fTable_Si[225, 2] := 3.57767;
    fTable_Si[226, 0] := 103.350; fTable_Si[226, 1] := -1.24200; fTable_Si[226, 2] := 3.56029;
    fTable_Si[227, 0] := 103.430; fTable_Si[227, 1] := -1.23327; fTable_Si[227, 2] := 3.47903;
    fTable_Si[228, 0] := 103.450; fTable_Si[228, 1] := -1.26147; fTable_Si[228, 2] := 3.44200;
    fTable_Si[229, 0] := 103.550; fTable_Si[229, 1] := -1.32267; fTable_Si[229, 2] := 3.37538;
    fTable_Si[230, 0] := 103.600; fTable_Si[230, 1] := -1.36022; fTable_Si[230, 2] := 3.35329;
    fTable_Si[231, 0] := 103.620; fTable_Si[231, 1] := -1.37658; fTable_Si[231, 2] := 3.35242;
    fTable_Si[232, 0] := 103.700; fTable_Si[232, 1] := -1.42690; fTable_Si[232, 2] := 3.33036;
    fTable_Si[233, 0] := 103.800; fTable_Si[233, 1] := -1.48061; fTable_Si[233, 2] := 3.33205;
    fTable_Si[234, 0] := 103.880; fTable_Si[234, 1] := -1.50969; fTable_Si[234, 2] := 3.33940;
    fTable_Si[235, 0] := 104.000; fTable_Si[235, 1] := -1.53630; fTable_Si[235, 2] := 3.33472;
    fTable_Si[236, 0] := 104.100; fTable_Si[236, 1] := -1.56167; fTable_Si[236, 2] := 3.31576;
    fTable_Si[237, 0] := 104.220; fTable_Si[237, 1] := -1.62193; fTable_Si[237, 2] := 3.27368;
    fTable_Si[238, 0] := 104.280; fTable_Si[238, 1] := -1.65400; fTable_Si[238, 2] := 3.27417;
    fTable_Si[239, 0] := 104.430; fTable_Si[239, 1] := -1.72694; fTable_Si[239, 2] := 3.28606;
    fTable_Si[240, 0] := 104.470; fTable_Si[240, 1] := -1.75387; fTable_Si[240, 2] := 3.27978;
    fTable_Si[241, 0] := 104.500; fTable_Si[241, 1] := -1.76829; fTable_Si[241, 2] := 3.28791;
    fTable_Si[242, 0] := 104.530; fTable_Si[242, 1] := -1.78693; fTable_Si[242, 2] := 3.28885;
    fTable_Si[243, 0] := 104.570; fTable_Si[243, 1] := -1.80294; fTable_Si[243, 2] := 3.29751;
    fTable_Si[244, 0] := 104.650; fTable_Si[244, 1] := -1.83679; fTable_Si[244, 2] := 3.30856;
    fTable_Si[245, 0] := 104.730; fTable_Si[245, 1] := -1.87270; fTable_Si[245, 2] := 3.30556;
    fTable_Si[246, 0] := 104.750; fTable_Si[246, 1] := -1.88124; fTable_Si[246, 2] := 3.31109;
    fTable_Si[247, 0] := 104.800; fTable_Si[247, 1] := -1.90801; fTable_Si[247, 2] := 3.30176;
    fTable_Si[248, 0] := 104.900; fTable_Si[248, 1] := -1.98706; fTable_Si[248, 2] := 3.33116;
    fTable_Si[249, 0] := 104.930; fTable_Si[249, 1] := -2.00067; fTable_Si[249, 2] := 3.33359;
    fTable_Si[250, 0] := 104.950; fTable_Si[250, 1] := -2.00298; fTable_Si[250, 2] := 3.34991;
    fTable_Si[251, 0] := 105.030; fTable_Si[251, 1] := -2.04570; fTable_Si[251, 2] := 3.36298;
    fTable_Si[252, 0] := 105.150; fTable_Si[252, 1] := -2.11934; fTable_Si[252, 2] := 3.39504;
    fTable_Si[253, 0] := 105.180; fTable_Si[253, 1] := -2.13949; fTable_Si[253, 2] := 3.40977;
    fTable_Si[254, 0] := 105.250; fTable_Si[254, 1] := -2.17952; fTable_Si[254, 2] := 3.43515;
    fTable_Si[255, 0] := 105.320; fTable_Si[255, 1] := -2.21343; fTable_Si[255, 2] := 3.47153;
    fTable_Si[256, 0] := 105.350; fTable_Si[256, 1] := -2.23848; fTable_Si[256, 2] := 3.47688;
    fTable_Si[257, 0] := 105.430; fTable_Si[257, 1] := -2.28483; fTable_Si[257, 2] := 3.52378;
    fTable_Si[258, 0] := 105.500; fTable_Si[258, 1] := -2.32999; fTable_Si[258, 2] := 3.56457;
    fTable_Si[259, 0] := 105.550; fTable_Si[259, 1] := -2.35832; fTable_Si[259, 2] := 3.60198;
    fTable_Si[260, 0] := 105.600; fTable_Si[260, 1] := -2.38578; fTable_Si[260, 2] := 3.64781;
    fTable_Si[261, 0] := 105.630; fTable_Si[261, 1] := -2.39089; fTable_Si[261, 2] := 3.66569;
    fTable_Si[262, 0] := 105.750; fTable_Si[262, 1] := -2.44861; fTable_Si[262, 2] := 3.77644;
    fTable_Si[263, 0] := 105.780; fTable_Si[263, 1] := -2.45326; fTable_Si[263, 2] := 3.79743;
    fTable_Si[264, 0] := 105.850; fTable_Si[264, 1] := -2.48245; fTable_Si[264, 2] := 3.88408;
    fTable_Si[265, 0] := 105.870; fTable_Si[265, 1] := -2.48052; fTable_Si[265, 2] := 3.91584;
    fTable_Si[266, 0] := 105.970; fTable_Si[266, 1] := -2.42689; fTable_Si[266, 2] := 4.01616;
    fTable_Si[267, 0] := 106.030; fTable_Si[267, 1] := -2.39972; fTable_Si[267, 2] := 4.04717;
    fTable_Si[268, 0] := 106.070; fTable_Si[268, 1] := -2.38240; fTable_Si[268, 2] := 4.06604;
    fTable_Si[269, 0] := 106.100; fTable_Si[269, 1] := -2.37398; fTable_Si[269, 2] := 4.06874;
    fTable_Si[270, 0] := 106.230; fTable_Si[270, 1] := -2.38361; fTable_Si[270, 2] := 4.11947;
    fTable_Si[271, 0] := 106.270; fTable_Si[271, 1] := -2.37996; fTable_Si[271, 2] := 4.15308;
    fTable_Si[272, 0] := 106.320; fTable_Si[272, 1] := -2.37462; fTable_Si[272, 2] := 4.16809;
    fTable_Si[273, 0] := 106.400; fTable_Si[273, 1] := -2.36004; fTable_Si[273, 2] := 4.21391;
    fTable_Si[274, 0] := 106.430; fTable_Si[274, 1] := -2.36196; fTable_Si[274, 2] := 4.22064;
    fTable_Si[275, 0] := 106.450; fTable_Si[275, 1] := -2.36509; fTable_Si[275, 2] := 4.23983;
    fTable_Si[276, 0] := 106.550; fTable_Si[276, 1] := -2.33925; fTable_Si[276, 2] := 4.28215;
    fTable_Si[277, 0] := 106.620; fTable_Si[277, 1] := -2.33379; fTable_Si[277, 2] := 4.30894;
    fTable_Si[278, 0] := 106.650; fTable_Si[278, 1] := -2.33507; fTable_Si[278, 2] := 4.32546;
    fTable_Si[279, 0] := 106.700; fTable_Si[279, 1] := -2.32865; fTable_Si[279, 2] := 4.34622;
    fTable_Si[280, 0] := 106.750; fTable_Si[280, 1] := -2.32543; fTable_Si[280, 2] := 4.37918;
    fTable_Si[281, 0] := 106.800; fTable_Si[281, 1] := -2.31100; fTable_Si[281, 2] := 4.39528;
    fTable_Si[282, 0] := 106.870; fTable_Si[282, 1] := -2.30275; fTable_Si[282, 2] := 4.43789;
    fTable_Si[283, 0] := 106.920; fTable_Si[283, 1] := -2.28031; fTable_Si[283, 2] := 4.45074;
    fTable_Si[284, 0] := 106.970; fTable_Si[284, 1] := -2.27262; fTable_Si[284, 2] := 4.47446;
    fTable_Si[285, 0] := 107.000; fTable_Si[285, 1] := -2.25035; fTable_Si[285, 2] := 4.47193;
    fTable_Si[286, 0] := 107.150; fTable_Si[286, 1] := -2.24976; fTable_Si[286, 2] := 4.52075;
    fTable_Si[287, 0] := 107.170; fTable_Si[287, 1] := -2.23267; fTable_Si[287, 2] := 4.52195;
    fTable_Si[288, 0] := 107.200; fTable_Si[288, 1] := -2.22431; fTable_Si[288, 2] := 4.53560;
    fTable_Si[289, 0] := 107.280; fTable_Si[289, 1] := -2.22372; fTable_Si[289, 2] := 4.53468;
    fTable_Si[290, 0] := 107.300; fTable_Si[290, 1] := -2.22218; fTable_Si[290, 2] := 4.54692;
    fTable_Si[291, 0] := 107.320; fTable_Si[291, 1] := -2.21789; fTable_Si[291, 2] := 4.54827;
    fTable_Si[292, 0] := 107.350; fTable_Si[292, 1] := -2.21747; fTable_Si[292, 2] := 4.55993;
    fTable_Si[293, 0] := 107.400; fTable_Si[293, 1] := -2.22568; fTable_Si[293, 2] := 4.56521;
    fTable_Si[294, 0] := 107.420; fTable_Si[294, 1] := -2.21201; fTable_Si[294, 2] := 4.58499;
    fTable_Si[295, 0] := 107.500; fTable_Si[295, 1] := -2.21196; fTable_Si[295, 2] := 4.60002;
    fTable_Si[296, 0] := 107.530; fTable_Si[296, 1] := -2.21439; fTable_Si[296, 2] := 4.60834;
    fTable_Si[297, 0] := 107.550; fTable_Si[297, 1] := -2.21478; fTable_Si[297, 2] := 4.62406;
    fTable_Si[298, 0] := 107.580; fTable_Si[298, 1] := -2.20227; fTable_Si[298, 2] := 4.63210;
    fTable_Si[299, 0] := 107.600; fTable_Si[299, 1] := -2.20862; fTable_Si[299, 2] := 4.62922;
    fTable_Si[300, 0] := 107.620; fTable_Si[300, 1] := -2.19987; fTable_Si[300, 2] := 4.64804;
    fTable_Si[301, 0] := 107.670; fTable_Si[301, 1] := -2.19745; fTable_Si[301, 2] := 4.66695;
    fTable_Si[302, 0] := 107.730; fTable_Si[302, 1] := -2.18227; fTable_Si[302, 2] := 4.67472;
    fTable_Si[303, 0] := 107.750; fTable_Si[303, 1] := -2.19300; fTable_Si[303, 2] := 4.68717;
    fTable_Si[304, 0] := 107.850; fTable_Si[304, 1] := -2.17068; fTable_Si[304, 2] := 4.70239;
    fTable_Si[305, 0] := 107.880; fTable_Si[305, 1] := -2.18424; fTable_Si[305, 2] := 4.71832;
    fTable_Si[306, 0] := 107.930; fTable_Si[306, 1] := -2.18294; fTable_Si[306, 2] := 4.73505;
    fTable_Si[307, 0] := 107.950; fTable_Si[307, 1] := -2.19199; fTable_Si[307, 2] := 4.75539;
    fTable_Si[308, 0] := 108.070; fTable_Si[308, 1] := -2.15772; fTable_Si[308, 2] := 4.79660;
    fTable_Si[309, 0] := 108.220; fTable_Si[309, 1] := -2.13084; fTable_Si[309, 2] := 4.82955;
    fTable_Si[310, 0] := 108.280; fTable_Si[310, 1] := -2.11240; fTable_Si[310, 2] := 4.85593;
    fTable_Si[311, 0] := 108.420; fTable_Si[311, 1] := -2.08897; fTable_Si[311, 2] := 4.88059;
    fTable_Si[312, 0] := 108.450; fTable_Si[312, 1] := -2.08958; fTable_Si[312, 2] := 4.88346;
    fTable_Si[313, 0] := 108.520; fTable_Si[313, 1] := -2.07611; fTable_Si[313, 2] := 4.91320;
    fTable_Si[314, 0] := 108.570; fTable_Si[314, 1] := -2.06068; fTable_Si[314, 2] := 4.91793;
    fTable_Si[315, 0] := 108.600; fTable_Si[315, 1] := -2.05985; fTable_Si[315, 2] := 4.93016;
    fTable_Si[316, 0] := 108.730; fTable_Si[316, 1] := -2.02793; fTable_Si[316, 2] := 4.92866;
    fTable_Si[317, 0] := 108.830; fTable_Si[317, 1] := -2.03087; fTable_Si[317, 2] := 4.94162;
    fTable_Si[318, 0] := 108.900; fTable_Si[318, 1] := -2.01993; fTable_Si[318, 2] := 4.96783;
    fTable_Si[319, 0] := 109.000; fTable_Si[319, 1] := -1.99875; fTable_Si[319, 2] := 4.97239;
    fTable_Si[320, 0] := 109.030; fTable_Si[320, 1] := -1.99361; fTable_Si[320, 2] := 4.97267;
    fTable_Si[321, 0] := 109.070; fTable_Si[321, 1] := -1.99579; fTable_Si[321, 2] := 4.95935;
    fTable_Si[322, 0] := 109.120; fTable_Si[322, 1] := -2.00066; fTable_Si[322, 2] := 4.97576;
    fTable_Si[323, 0] := 109.200; fTable_Si[323, 1] := -2.00421; fTable_Si[323, 2] := 4.98276;
    fTable_Si[324, 0] := 109.250; fTable_Si[324, 1] := -1.99981; fTable_Si[324, 2] := 4.99897;
    fTable_Si[325, 0] := 109.270; fTable_Si[325, 1] := -1.98698; fTable_Si[325, 2] := 4.98829;
    fTable_Si[326, 0] := 109.350; fTable_Si[326, 1] := -2.00603; fTable_Si[326, 2] := 4.99135;
    fTable_Si[327, 0] := 109.380; fTable_Si[327, 1] := -2.00850; fTable_Si[327, 2] := 4.98316;
    fTable_Si[328, 0] := 109.400; fTable_Si[328, 1] := -2.01211; fTable_Si[328, 2] := 4.99342;
    fTable_Si[329, 0] := 109.430; fTable_Si[329, 1] := -2.02183; fTable_Si[329, 2] := 4.98967;
    fTable_Si[330, 0] := 109.450; fTable_Si[330, 1] := -2.01515; fTable_Si[330, 2] := 5.00593;
    fTable_Si[331, 0] := 109.530; fTable_Si[331, 1] := -2.04292; fTable_Si[331, 2] := 5.01580;
    fTable_Si[332, 0] := 109.550; fTable_Si[332, 1] := -2.03376; fTable_Si[332, 2] := 5.03141;
    fTable_Si[333, 0] := 109.570; fTable_Si[333, 1] := -2.03838; fTable_Si[333, 2] := 5.02656;
    fTable_Si[334, 0] := 109.600; fTable_Si[334, 1] := -2.03677; fTable_Si[334, 2] := 5.04483;
    fTable_Si[335, 0] := 109.620; fTable_Si[335, 1] := -2.03705; fTable_Si[335, 2] := 5.03873;
    fTable_Si[336, 0] := 109.670; fTable_Si[336, 1] := -2.02773; fTable_Si[336, 2] := 5.05325;
    fTable_Si[337, 0] := 109.800; fTable_Si[337, 1] := -2.05572; fTable_Si[337, 2] := 5.08673;
    fTable_Si[338, 0] := 109.970; fTable_Si[338, 1] := -2.05841; fTable_Si[338, 2] := 5.12220;
    fTable_Si[339, 0] := 110.000; fTable_Si[339, 1] := -2.08477; fTable_Si[339, 2] := 5.13791;
    fTable_Si[340, 0] := 110.500; fTable_Si[340, 1] := -2.08318; fTable_Si[340, 2] := 5.28267;
    fTable_Si[341, 0] := 111.000; fTable_Si[341, 1] := -2.07105; fTable_Si[341, 2] := 5.45779;
    fTable_Si[342, 0] := 111.500; fTable_Si[342, 1] := -2.02987; fTable_Si[342, 2] := 5.61544;
    fTable_Si[343, 0] := 112.500; fTable_Si[343, 1] := -1.94845; fTable_Si[343, 2] := 5.85909;
    fTable_Si[344, 0] := 114.000; fTable_Si[344, 1] := -1.92517; fTable_Si[344, 2] := 6.16450;
    fTable_Si[345, 0] := 114.500; fTable_Si[345, 1] := -1.96395; fTable_Si[345, 2] := 6.33338;
    fTable_Si[346, 0] := 115.000; fTable_Si[346, 1] := -1.98987; fTable_Si[346, 2] := 6.51862;
    fTable_Si[347, 0] := 115.500; fTable_Si[347, 1] := -1.96320; fTable_Si[347, 2] := 6.72312;
    fTable_Si[348, 0] := 117.000; fTable_Si[348, 1] := -1.77809; fTable_Si[348, 2] := 7.40254;
    fTable_Si[349, 0] := 117.500; fTable_Si[349, 1] := -1.61173; fTable_Si[349, 2] := 7.59488;
    fTable_Si[350, 0] := 118.000; fTable_Si[350, 1] := -1.45934; fTable_Si[350, 2] := 7.77180;
    fTable_Si[351, 0] := 118.500; fTable_Si[351, 1] := -1.28616; fTable_Si[351, 2] := 7.87553;
    fTable_Si[352, 0] := 119.000; fTable_Si[352, 1] := -1.13984; fTable_Si[352, 2] := 8.02234;
    fTable_Si[353, 0] := 119.500; fTable_Si[353, 1] := -0.959918; fTable_Si[353, 2] := 8.05843;
    fTable_Si[354, 0] := 121.433; fTable_Si[354, 1] := -0.578394; fTable_Si[354, 2] := 8.42371;
    fTable_Si[355, 0] := 121.500; fTable_Si[355, 1] := -0.573231; fTable_Si[355, 2] := 8.43660;
    fTable_Si[356, 0] := 122.000; fTable_Si[356, 1] := -0.405651; fTable_Si[356, 2] := 8.51447;
    fTable_Si[357, 0] := 123.500; fTable_Si[357, 1] := -0.0264126; fTable_Si[357, 2] := 8.67192;
    fTable_Si[358, 0] := 124.000; fTable_Si[358, 1] := 0.0779155; fTable_Si[358, 2] := 8.69958;
    fTable_Si[359, 0] := 124.500; fTable_Si[359, 1] := 0.171345; fTable_Si[359, 2] := 8.77704;
    fTable_Si[360, 0] := 125.000; fTable_Si[360, 1] := 0.293945; fTable_Si[360, 2] := 8.78726;
    fTable_Si[361, 0] := 127.000; fTable_Si[361, 1] := 0.572464; fTable_Si[361, 2] := 9.00076;
    fTable_Si[362, 0] := 127.500; fTable_Si[362, 1] := 0.671836; fTable_Si[362, 2] := 9.04215;
    fTable_Si[363, 0] := 128.500; fTable_Si[363, 1] := 0.827038; fTable_Si[363, 2] := 9.19455;
    fTable_Si[364, 0] := 129.500; fTable_Si[364, 1] := 0.995074; fTable_Si[364, 2] := 9.33439;
    fTable_Si[365, 0] := 130.000; fTable_Si[365, 1] := 1.11832; fTable_Si[365, 2] := 9.43724;
    fTable_Si[366, 0] := 131.500; fTable_Si[366, 1] := 1.53131; fTable_Si[366, 2] := 9.68832;
    fTable_Si[367, 0] := 133.000; fTable_Si[367, 1] := 2.07611; fTable_Si[367, 2] := 9.80683;
    fTable_Si[368, 0] := 133.500; fTable_Si[368, 1] := 2.28741; fTable_Si[368, 2] := 9.78221;
    fTable_Si[369, 0] := 134.500; fTable_Si[369, 1] := 2.61972; fTable_Si[369, 2] := 9.60861;
    fTable_Si[370, 0] := 136.000; fTable_Si[370, 1] := 2.84736; fTable_Si[370, 2] := 9.24827;
    fTable_Si[371, 0] := 136.500; fTable_Si[371, 1] := 2.87943; fTable_Si[371, 2] := 9.17385;
    fTable_Si[372, 0] := 137.000; fTable_Si[372, 1] := 2.87745; fTable_Si[372, 2] := 9.11857;
    fTable_Si[373, 0] := 137.500; fTable_Si[373, 1] := 2.85152; fTable_Si[373, 2] := 9.03612;
    fTable_Si[374, 0] := 139.500; fTable_Si[374, 1] := 2.83348; fTable_Si[374, 2] := 9.09883;
    fTable_Si[375, 0] := 140.000; fTable_Si[375, 1] := 2.84307; fTable_Si[375, 2] := 9.12631;
    fTable_Si[376, 0] := 140.500; fTable_Si[376, 1] := 2.88384; fTable_Si[376, 2] := 9.18357;
    fTable_Si[377, 0] := 141.500; fTable_Si[377, 1] := 3.00310; fTable_Si[377, 2] := 9.19764;
    fTable_Si[378, 0] := 142.000; fTable_Si[378, 1] := 3.03093; fTable_Si[378, 2] := 9.17508;
    fTable_Si[379, 0] := 142.500; fTable_Si[379, 1] := 3.03358; fTable_Si[379, 2] := 9.18522;
    fTable_Si[380, 0] := 143.000; fTable_Si[380, 1] := 3.03374; fTable_Si[380, 2] := 9.17393;
    fTable_Si[381, 0] := 144.000; fTable_Si[381, 1] := 3.03215; fTable_Si[381, 2] := 9.32209;
    fTable_Si[382, 0] := 145.000; fTable_Si[382, 1] := 3.09900; fTable_Si[382, 2] := 9.41818;
    fTable_Si[383, 0] := 145.500; fTable_Si[383, 1] := 3.16288; fTable_Si[383, 2] := 9.49844;
    fTable_Si[384, 0] := 146.000; fTable_Si[384, 1] := 3.22259; fTable_Si[384, 2] := 9.51997;
    fTable_Si[385, 0] := 146.500; fTable_Si[385, 1] := 3.28049; fTable_Si[385, 2] := 9.57995;
    fTable_Si[386, 0] := 147.000; fTable_Si[386, 1] := 3.34172; fTable_Si[386, 2] := 9.60862;
    fTable_Si[387, 0] := 147.500; fTable_Si[387, 1] := 3.41479; fTable_Si[387, 2] := 9.66258;
    fTable_Si[388, 0] := 148.000; fTable_Si[388, 1] := 3.48151; fTable_Si[388, 2] := 9.67350;
    fTable_Si[389, 0] := 148.500; fTable_Si[389, 1] := 3.56199; fTable_Si[389, 2] := 9.71113;
    fTable_Si[390, 0] := 149.500; fTable_Si[390, 1] := 3.68256; fTable_Si[390, 2] := 9.71835;
    fTable_Si[391, 0] := 150.000; fTable_Si[391, 1] := 3.70254; fTable_Si[391, 2] := 9.69979;
    fTable_Si[392, 0] := 150.500; fTable_Si[392, 1] := 3.68373; fTable_Si[392, 2] := 9.74096;
    fTable_Si[393, 0] := 151.000; fTable_Si[393, 1] := 3.69207; fTable_Si[393, 2] := 9.84710;
    fTable_Si[394, 0] := 151.500; fTable_Si[394, 1] := 3.76904; fTable_Si[394, 2] := 10.0037;
    fTable_Si[395, 0] := 152.000; fTable_Si[395, 1] := 3.94900; fTable_Si[395, 2] := 10.1180;
    fTable_Si[396, 0] := 152.500; fTable_Si[396, 1] := 4.15147; fTable_Si[396, 2] := 10.1431;
    fTable_Si[397, 0] := 153.500; fTable_Si[397, 1] := 4.47402; fTable_Si[397, 2] := 9.96424;
    fTable_Si[398, 0] := 154.500; fTable_Si[398, 1] := 4.52214; fTable_Si[398, 2] := 9.69132;
    fTable_Si[399, 0] := 155.000; fTable_Si[399, 1] := 4.47788; fTable_Si[399, 2] := 9.64167;
    fTable_Si[400, 0] := 155.500; fTable_Si[400, 1] := 4.41664; fTable_Si[400, 2] := 9.63644;
    fTable_Si[401, 0] := 156.000; fTable_Si[401, 1] := 4.38177; fTable_Si[401, 2] := 9.66128;
    fTable_Si[402, 0] := 156.500; fTable_Si[402, 1] := 4.35929; fTable_Si[402, 2] := 9.73288;
    fTable_Si[403, 0] := 157.500; fTable_Si[403, 1] := 4.39020; fTable_Si[403, 2] := 9.79855;
    fTable_Si[404, 0] := 158.000; fTable_Si[404, 1] := 4.36737; fTable_Si[404, 2] := 9.87036;
    fTable_Si[405, 0] := 158.500; fTable_Si[405, 1] := 4.42951; fTable_Si[405, 2] := 9.99628;
    fTable_Si[406, 0] := 159.000; fTable_Si[406, 1] := 4.48663; fTable_Si[406, 2] := 9.99841;
    fTable_Si[407, 0] := 160.000; fTable_Si[407, 1] := 4.57954; fTable_Si[407, 2] := 10.1071;
    fTable_Si[408, 0] := 162.500; fTable_Si[408, 1] := 4.84589; fTable_Si[408, 2] := 10.5019;
    fTable_Si[409, 0] := 163.500; fTable_Si[409, 1] := 5.05409; fTable_Si[409, 2] := 10.6336;
    fTable_Si[410, 0] := 164.500; fTable_Si[410, 1] := 5.27583; fTable_Si[410, 2] := 10.7324;
    fTable_Si[411, 0] := 165.500; fTable_Si[411, 1] := 5.50795; fTable_Si[411, 2] := 10.7656;
    fTable_Si[412, 0] := 166.500; fTable_Si[412, 1] := 5.73389; fTable_Si[412, 2] := 10.8239;
    fTable_Si[413, 0] := 167.000; fTable_Si[413, 1] := 5.79695; fTable_Si[413, 2] := 10.7800;
    fTable_Si[414, 0] := 167.500; fTable_Si[414, 1] := 5.86489; fTable_Si[414, 2] := 10.9015;
    fTable_Si[415, 0] := 169.000; fTable_Si[415, 1] := 6.35522; fTable_Si[415, 2] := 10.9520;
    fTable_Si[416, 0] := 170.000; fTable_Si[416, 1] := 6.66644; fTable_Si[416, 2] := 10.9210;
    fTable_Si[417, 0] := 171.500; fTable_Si[417, 1] := 7.13398; fTable_Si[417, 2] := 10.7554;
    fTable_Si[418, 0] := 172.000; fTable_Si[418, 1] := 7.24279; fTable_Si[418, 2] := 10.5495;
    fTable_Si[419, 0] := 172.500; fTable_Si[419, 1] := 7.29281; fTable_Si[419, 2] := 10.5369;
    fTable_Si[420, 0] := 173.000; fTable_Si[420, 1] := 7.38343; fTable_Si[420, 2] := 10.4391;
    fTable_Si[421, 0] := 173.500; fTable_Si[421, 1] := 7.52303; fTable_Si[421, 2] := 10.4208;
    fTable_Si[422, 0] := 174.000; fTable_Si[422, 1] := 7.60600; fTable_Si[422, 2] := 10.1923;
    fTable_Si[423, 0] := 174.500; fTable_Si[423, 1] := 7.64212; fTable_Si[423, 2] := 10.1249;
    fTable_Si[424, 0] := 175.000; fTable_Si[424, 1] := 7.66842; fTable_Si[424, 2] := 9.98038;
    fTable_Si[425, 0] := 176.000; fTable_Si[425, 1] := 7.68591; fTable_Si[425, 2] := 9.82584;
    fTable_Si[426, 0] := 176.500; fTable_Si[426, 1] := 7.67332; fTable_Si[426, 2] := 9.72546;
    fTable_Si[427, 0] := 177.000; fTable_Si[427, 1] := 7.68563; fTable_Si[427, 2] := 9.66145;
    fTable_Si[428, 0] := 178.000; fTable_Si[428, 1] := 7.67511; fTable_Si[428, 2] := 9.60542;
    fTable_Si[429, 0] := 178.500; fTable_Si[429, 1] := 7.69740; fTable_Si[429, 2] := 9.51565;
    fTable_Si[430, 0] := 179.000; fTable_Si[430, 1] := 7.64095; fTable_Si[430, 2] := 9.49283;
    fTable_Si[431, 0] := 179.500; fTable_Si[431, 1] := 7.63925; fTable_Si[431, 2] := 9.43704;
    fTable_Si[432, 0] := 179.990; fTable_Si[432, 1] := 7.55398; fTable_Si[432, 2] := 9.49765;
    fTable_Si[433, 0] := 182.901; fTable_Si[433, 1] := 7.85149; fTable_Si[433, 2] := 9.42072;
    fTable_Si[434, 0] := 185.859; fTable_Si[434, 1] := 7.94847; fTable_Si[434, 2] := 9.34442;
    fTable_Si[435, 0] := 188.866; fTable_Si[435, 1] := 8.10574; fTable_Si[435, 2] := 9.26640;
    fTable_Si[436, 0] := 191.920; fTable_Si[436, 1] := 8.27005; fTable_Si[436, 2] := 9.17918;
    fTable_Si[437, 0] := 195.025; fTable_Si[437, 1] := 8.43202; fTable_Si[437, 2] := 9.09278;
    fTable_Si[438, 0] := 198.179; fTable_Si[438, 1] := 8.59128; fTable_Si[438, 2] := 9.00719;
    fTable_Si[439, 0] := 201.384; fTable_Si[439, 1] := 8.74251; fTable_Si[439, 2] := 8.92241;
    fTable_Si[440, 0] := 204.641; fTable_Si[440, 1] := 8.88646; fTable_Si[440, 2] := 8.85010;
    fTable_Si[441, 0] := 207.951; fTable_Si[441, 1] := 9.03960; fTable_Si[441, 2] := 8.78533;
    fTable_Si[442, 0] := 211.315; fTable_Si[442, 1] := 9.19861; fTable_Si[442, 2] := 8.72104;
    fTable_Si[443, 0] := 214.733; fTable_Si[443, 1] := 9.36085; fTable_Si[443, 2] := 8.65722;
    fTable_Si[444, 0] := 218.206; fTable_Si[444, 1] := 9.53668; fTable_Si[444, 2] := 8.59386;
    fTable_Si[445, 0] := 221.735; fTable_Si[445, 1] := 9.72509; fTable_Si[445, 2] := 8.52313;
    fTable_Si[446, 0] := 225.322; fTable_Si[446, 1] := 9.90451; fTable_Si[446, 2] := 8.41115;
    fTable_Si[447, 0] := 228.966; fTable_Si[447, 1] := 10.0644; fTable_Si[447, 2] := 8.30065;
    fTable_Si[448, 0] := 232.669; fTable_Si[448, 1] := 10.2142; fTable_Si[448, 2] := 8.19159;
    fTable_Si[449, 0] := 236.432; fTable_Si[449, 1] := 10.3574; fTable_Si[449, 2] := 8.08397;
    fTable_Si[450, 0] := 240.257; fTable_Si[450, 1] := 10.4958; fTable_Si[450, 2] := 7.97776;
    fTable_Si[451, 0] := 244.143; fTable_Si[451, 1] := 10.6314; fTable_Si[451, 2] := 7.87295;
    fTable_Si[452, 0] := 248.091; fTable_Si[452, 1] := 10.7716; fTable_Si[452, 2] := 7.76952;
    fTable_Si[453, 0] := 252.104; fTable_Si[453, 1] := 10.9063; fTable_Si[453, 2] := 7.65024;
    fTable_Si[454, 0] := 256.182; fTable_Si[454, 1] := 11.0283; fTable_Si[454, 2] := 7.53005;
    fTable_Si[455, 0] := 260.325; fTable_Si[455, 1] := 11.1426; fTable_Si[455, 2] := 7.41174;
    fTable_Si[456, 0] := 264.536; fTable_Si[456, 1] := 11.2509; fTable_Si[456, 2] := 7.29529;
    fTable_Si[457, 0] := 268.814; fTable_Si[457, 1] := 11.3543; fTable_Si[457, 2] := 7.18067;
    fTable_Si[458, 0] := 273.162; fTable_Si[458, 1] := 11.4535; fTable_Si[458, 2] := 7.06784;
    fTable_Si[459, 0] := 277.580; fTable_Si[459, 1] := 11.5489; fTable_Si[459, 2] := 6.95680;
    fTable_Si[460, 0] := 282.070; fTable_Si[460, 1] := 11.6411; fTable_Si[460, 2] := 6.84750;
    fTable_Si[461, 0] := 286.632; fTable_Si[461, 1] := 11.7306; fTable_Si[461, 2] := 6.73991;
    fTable_Si[462, 0] := 291.268; fTable_Si[462, 1] := 11.8181; fTable_Si[462, 2] := 6.63402;
    fTable_Si[463, 0] := 295.979; fTable_Si[463, 1] := 11.9057; fTable_Si[463, 2] := 6.52979;
    fTable_Si[464, 0] := 300.767; fTable_Si[464, 1] := 11.9918; fTable_Si[464, 2] := 6.42157;
    fTable_Si[465, 0] := 305.631; fTable_Si[465, 1] := 12.0733; fTable_Si[465, 2] := 6.31071;
    fTable_Si[466, 0] := 310.575; fTable_Si[466, 1] := 12.1486; fTable_Si[466, 2] := 6.20175;
    fTable_Si[467, 0] := 315.598; fTable_Si[467, 1] := 12.2203; fTable_Si[467, 2] := 6.09469;
    fTable_Si[468, 0] := 320.702; fTable_Si[468, 1] := 12.2889; fTable_Si[468, 2] := 5.98947;
    fTable_Si[469, 0] := 325.890; fTable_Si[469, 1] := 12.3551; fTable_Si[469, 2] := 5.88607;
    fTable_Si[470, 0] := 331.161; fTable_Si[470, 1] := 12.4191; fTable_Si[470, 2] := 5.78445;
    fTable_Si[471, 0] := 336.517; fTable_Si[471, 1] := 12.4812; fTable_Si[471, 2] := 5.68459;
    fTable_Si[472, 0] := 341.960; fTable_Si[472, 1] := 12.5420; fTable_Si[472, 2] := 5.58645;
    fTable_Si[473, 0] := 347.491; fTable_Si[473, 1] := 12.6018; fTable_Si[473, 2] := 5.49000;
    fTable_Si[474, 0] := 353.111; fTable_Si[474, 1] := 12.6614; fTable_Si[474, 2] := 5.39523;
    fTable_Si[475, 0] := 358.822; fTable_Si[475, 1] := 12.7222; fTable_Si[475, 2] := 5.30208;
    fTable_Si[476, 0] := 364.626; fTable_Si[476, 1] := 12.7889; fTable_Si[476, 2] := 5.21055;
    fTable_Si[477, 0] := 370.523; fTable_Si[477, 1] := 12.8576; fTable_Si[477, 2] := 5.10056;
    fTable_Si[478, 0] := 376.516; fTable_Si[478, 1] := 12.9142; fTable_Si[478, 2] := 4.98768;
    fTable_Si[479, 0] := 382.606; fTable_Si[479, 1] := 12.9608; fTable_Si[479, 2] := 4.87731;
    fTable_Si[480, 0] := 388.795; fTable_Si[480, 1] := 13.0027; fTable_Si[480, 2] := 4.76937;
    fTable_Si[481, 0] := 395.083; fTable_Si[481, 1] := 13.0407; fTable_Si[481, 2] := 4.66382;
    fTable_Si[482, 0] := 401.473; fTable_Si[482, 1] := 13.0753; fTable_Si[482, 2] := 4.56061;
    fTable_Si[483, 0] := 407.967; fTable_Si[483, 1] := 13.1069; fTable_Si[483, 2] := 4.45967;
    fTable_Si[484, 0] := 414.565; fTable_Si[484, 1] := 13.1360; fTable_Si[484, 2] := 4.36098;
    fTable_Si[485, 0] := 421.270; fTable_Si[485, 1] := 13.1628; fTable_Si[485, 2] := 4.26447;
    fTable_Si[486, 0] := 428.084; fTable_Si[486, 1] := 13.1876; fTable_Si[486, 2] := 4.17009;
    fTable_Si[487, 0] := 435.008; fTable_Si[487, 1] := 13.2107; fTable_Si[487, 2] := 4.07781;
    fTable_Si[488, 0] := 442.044; fTable_Si[488, 1] := 13.2322; fTable_Si[488, 2] := 3.98756;
    fTable_Si[489, 0] := 449.194; fTable_Si[489, 1] := 13.2527; fTable_Si[489, 2] := 3.89931;
    fTable_Si[490, 0] := 456.459; fTable_Si[490, 1] := 13.2727; fTable_Si[490, 2] := 3.81302;
    fTable_Si[491, 0] := 463.842; fTable_Si[491, 1] := 13.2933; fTable_Si[491, 2] := 3.72727;
    fTable_Si[492, 0] := 471.344; fTable_Si[492, 1] := 13.3117; fTable_Si[492, 2] := 3.63809;
    fTable_Si[493, 0] := 478.968; fTable_Si[493, 1] := 13.3260; fTable_Si[493, 2] := 3.55105;
    fTable_Si[494, 0] := 486.715; fTable_Si[494, 1] := 13.3375; fTable_Si[494, 2] := 3.46608;
    fTable_Si[495, 0] := 494.587; fTable_Si[495, 1] := 13.3472; fTable_Si[495, 2] := 3.38316;
    fTable_Si[496, 0] := 502.587; fTable_Si[496, 1] := 13.3552; fTable_Si[496, 2] := 3.30221;
    fTable_Si[497, 0] := 510.715; fTable_Si[497, 1] := 13.3617; fTable_Si[497, 2] := 3.22320;
    fTable_Si[498, 0] := 518.976; fTable_Si[498, 1] := 13.3670; fTable_Si[498, 2] := 3.14609;
    fTable_Si[499, 0] := 527.370; fTable_Si[499, 1] := 13.3711; fTable_Si[499, 2] := 3.07081;
    fTable_Si[500, 0] := 535.900; fTable_Si[500, 1] := 13.3742; fTable_Si[500, 2] := 2.99734;
    fTable_Si[501, 0] := 544.567; fTable_Si[501, 1] := 13.3764; fTable_Si[501, 2] := 2.92563;
    fTable_Si[502, 0] := 553.375; fTable_Si[502, 1] := 13.3779; fTable_Si[502, 2] := 2.85563;
    fTable_Si[503, 0] := 562.326; fTable_Si[503, 1] := 13.3789; fTable_Si[503, 2] := 2.78730;
    fTable_Si[504, 0] := 571.421; fTable_Si[504, 1] := 13.3797; fTable_Si[504, 2] := 2.72061;
    fTable_Si[505, 0] := 580.663; fTable_Si[505, 1] := 13.3815; fTable_Si[505, 2] := 2.65552;
    fTable_Si[506, 0] := 590.055; fTable_Si[506, 1] := 13.3832; fTable_Si[506, 2] := 2.58813;
    fTable_Si[507, 0] := 599.599; fTable_Si[507, 1] := 13.3823; fTable_Si[507, 2] := 2.52006;
    fTable_Si[508, 0] := 609.297; fTable_Si[508, 1] := 13.3786; fTable_Si[508, 2] := 2.45378;
    fTable_Si[509, 0] := 619.151; fTable_Si[509, 1] := 13.3731; fTable_Si[509, 2] := 2.38925;
    fTable_Si[510, 0] := 629.166; fTable_Si[510, 1] := 13.3663; fTable_Si[510, 2] := 2.32641;
    fTable_Si[511, 0] := 639.342; fTable_Si[511, 1] := 13.3582; fTable_Si[511, 2] := 2.26522;
    fTable_Si[512, 0] := 649.683; fTable_Si[512, 1] := 13.3491; fTable_Si[512, 2] := 2.20565;
    fTable_Si[513, 0] := 660.191; fTable_Si[513, 1] := 13.3390; fTable_Si[513, 2] := 2.14764;
    fTable_Si[514, 0] := 670.869; fTable_Si[514, 1] := 13.3278; fTable_Si[514, 2] := 2.09115;
    fTable_Si[515, 0] := 681.720; fTable_Si[515, 1] := 13.3158; fTable_Si[515, 2] := 2.03616;
    fTable_Si[516, 0] := 692.746; fTable_Si[516, 1] := 13.3006; fTable_Si[516, 2] := 1.98261;
    fTable_Si[517, 0] := 703.951; fTable_Si[517, 1] := 13.2845; fTable_Si[517, 2] := 1.93392;
    fTable_Si[518, 0] := 715.336; fTable_Si[518, 1] := 13.2706; fTable_Si[518, 2] := 1.88812;
    fTable_Si[519, 0] := 726.906; fTable_Si[519, 1] := 13.2578; fTable_Si[519, 2] := 1.84339;
    fTable_Si[520, 0] := 738.664; fTable_Si[520, 1] := 13.2453; fTable_Si[520, 2] := 1.79973;
    fTable_Si[521, 0] := 750.611; fTable_Si[521, 1] := 13.2332; fTable_Si[521, 2] := 1.75710;
    fTable_Si[522, 0] := 762.751; fTable_Si[522, 1] := 13.2215; fTable_Si[522, 2] := 1.71548;
    fTable_Si[523, 0] := 775.088; fTable_Si[523, 1] := 13.2102; fTable_Si[523, 2] := 1.67484;
    fTable_Si[524, 0] := 787.625; fTable_Si[524, 1] := 13.1996; fTable_Si[524, 2] := 1.63517;
    fTable_Si[525, 0] := 800.364; fTable_Si[525, 1] := 13.1912; fTable_Si[525, 2] := 1.59508;
    fTable_Si[526, 0] := 813.309; fTable_Si[526, 1] := 13.1807; fTable_Si[526, 2] := 1.55256;
    fTable_Si[527, 0] := 826.464; fTable_Si[527, 1] := 13.1685; fTable_Si[527, 2] := 1.51118;
    fTable_Si[528, 0] := 839.831; fTable_Si[528, 1] := 13.1555; fTable_Si[528, 2] := 1.47089;
    fTable_Si[529, 0] := 853.415; fTable_Si[529, 1] := 13.1418; fTable_Si[529, 2] := 1.43168;
    fTable_Si[530, 0] := 867.218; fTable_Si[530, 1] := 13.1278; fTable_Si[530, 2] := 1.39352;
    fTable_Si[531, 0] := 881.245; fTable_Si[531, 1] := 13.1136; fTable_Si[531, 2] := 1.35637;
    fTable_Si[532, 0] := 895.498; fTable_Si[532, 1] := 13.1001; fTable_Si[532, 2] := 1.32021;
    fTable_Si[533, 0] := 909.982; fTable_Si[533, 1] := 13.0874; fTable_Si[533, 2] := 1.28196;
    fTable_Si[534, 0] := 924.700; fTable_Si[534, 1] := 13.0717; fTable_Si[534, 2] := 1.24308;
    fTable_Si[535, 0] := 939.656; fTable_Si[535, 1] := 13.0542; fTable_Si[535, 2] := 1.20538;
    fTable_Si[536, 0] := 954.855; fTable_Si[536, 1] := 13.0353; fTable_Si[536, 2] := 1.16882;
    fTable_Si[537, 0] := 970.299; fTable_Si[537, 1] := 13.0154; fTable_Si[537, 2] := 1.13337;
    fTable_Si[538, 0] := 985.992; fTable_Si[538, 1] := 12.9946; fTable_Si[538, 2] := 1.09899;
    fTable_Si[539, 0] := 1001.94; fTable_Si[539, 1] := 12.9729; fTable_Si[539, 2] := 1.06561;
    fTable_Si[540, 0] := 1018.15; fTable_Si[540, 1] := 12.9502; fTable_Si[540, 2] := 1.03318;
    fTable_Si[541, 0] := 1034.61; fTable_Si[541, 1] := 12.9266; fTable_Si[541, 2] := 1.00174;
    fTable_Si[542, 0] := 1051.35; fTable_Si[542, 1] := 12.9020; fTable_Si[542, 2] := 0.971249;
    fTable_Si[543, 0] := 1068.35; fTable_Si[543, 1] := 12.8761; fTable_Si[543, 2] := 0.941688;
    fTable_Si[544, 0] := 1085.63; fTable_Si[544, 1] := 12.8487; fTable_Si[544, 2] := 0.913028;
    fTable_Si[545, 0] := 1103.19; fTable_Si[545, 1] := 12.8192; fTable_Si[545, 2] := 0.887547;
    fTable_Si[546, 0] := 1121.03; fTable_Si[546, 1] := 12.7911; fTable_Si[546, 2] := 0.864407;
    fTable_Si[547, 0] := 1139.17; fTable_Si[547, 1] := 12.7632; fTable_Si[547, 2] := 0.841817;
    fTable_Si[548, 0] := 1157.59; fTable_Si[548, 1] := 12.7350; fTable_Si[548, 2] := 0.819826;
    fTable_Si[549, 0] := 1176.31; fTable_Si[549, 1] := 12.7063; fTable_Si[549, 2] := 0.798411;
    fTable_Si[550, 0] := 1195.34; fTable_Si[550, 1] := 12.6771; fTable_Si[550, 2] := 0.777531;
    fTable_Si[551, 0] := 1214.67; fTable_Si[551, 1] := 12.6470; fTable_Si[551, 2] := 0.757139;
    fTable_Si[552, 0] := 1234.32; fTable_Si[552, 1] := 12.6159; fTable_Si[552, 2] := 0.737234;
    fTable_Si[553, 0] := 1254.28; fTable_Si[553, 1] := 12.5837; fTable_Si[553, 2] := 0.717856;
    fTable_Si[554, 0] := 1274.57; fTable_Si[554, 1] := 12.5503; fTable_Si[554, 2] := 0.698989;
    fTable_Si[555, 0] := 1295.19; fTable_Si[555, 1] := 12.5156; fTable_Si[555, 2] := 0.680609;
    fTable_Si[556, 0] := 1316.13; fTable_Si[556, 1] := 12.4792; fTable_Si[556, 2] := 0.662552;
    fTable_Si[557, 0] := 1337.42; fTable_Si[557, 1] := 12.4409; fTable_Si[557, 2] := 0.644954;
    fTable_Si[558, 0] := 1359.05; fTable_Si[558, 1] := 12.4006; fTable_Si[558, 2] := 0.627806;
    fTable_Si[559, 0] := 1381.04; fTable_Si[559, 1] := 12.3579; fTable_Si[559, 2] := 0.611117;
    fTable_Si[560, 0] := 1403.37; fTable_Si[560, 1] := 12.3125; fTable_Si[560, 2] := 0.594814;
    fTable_Si[561, 0] := 1426.07; fTable_Si[561, 1] := 12.2640; fTable_Si[561, 2] := 0.578892;
    fTable_Si[562, 0] := 1449.14; fTable_Si[562, 1] := 12.2120; fTable_Si[562, 2] := 0.563357;
    fTable_Si[563, 0] := 1472.58; fTable_Si[563, 1] := 12.1559; fTable_Si[563, 2] := 0.548240;
    fTable_Si[564, 0] := 1496.39; fTable_Si[564, 1] := 12.0950; fTable_Si[564, 2] := 0.533519;
    fTable_Si[565, 0] := 1520.60; fTable_Si[565, 1] := 12.0284; fTable_Si[565, 2] := 0.518512;
    fTable_Si[566, 0] := 1545.19; fTable_Si[566, 1] := 11.9546; fTable_Si[566, 2] := 0.503884;
    fTable_Si[567, 0] := 1570.18; fTable_Si[567, 1] := 11.8721; fTable_Si[567, 2] := 0.489627;
    fTable_Si[568, 0] := 1595.58; fTable_Si[568, 1] := 11.7790; fTable_Si[568, 2] := 0.475781;
    fTable_Si[569, 0] := 1621.39; fTable_Si[569, 1] := 11.6727; fTable_Si[569, 2] := 0.462322;
    fTable_Si[570, 0] := 1647.61; fTable_Si[570, 1] := 11.5493; fTable_Si[570, 2] := 0.449240;
    fTable_Si[571, 0] := 1674.26; fTable_Si[571, 1] := 11.4029; fTable_Si[571, 2] := 0.436529;
    fTable_Si[572, 0] := 1701.34; fTable_Si[572, 1] := 11.2243; fTable_Si[572, 2] := 0.424180;
    fTable_Si[573, 0] := 1728.86; fTable_Si[573, 1] := 10.9982; fTable_Si[573, 2] := 0.412181;
    fTable_Si[574, 0] := 1756.82; fTable_Si[574, 1] := 10.6935; fTable_Si[574, 2] := 0.399995;
    fTable_Si[575, 0] := 1785.24; fTable_Si[575, 1] := 10.2377; fTable_Si[575, 2] := 0.388066;
    fTable_Si[576, 0] := 1814.11; fTable_Si[576, 1] := 9.37942; fTable_Si[576, 2] := 0.376400;
    fTable_Si[577, 0] := 1815; fTable_Si[577, 1] := 9.33435; fTable_Si[577, 2] := 0.376049;
    fTable_Si[578, 0] := 1838.80; fTable_Si[578, 1] := 2.82013; fTable_Si[578, 2] := 0.366843;
    fTable_Si[579, 0] := 1838.90; fTable_Si[579, 1] := 7.96957; fTable_Si[579, 2] := 4.15773;
    fTable_Si[580, 0] := 1839; fTable_Si[580, 1] := 2.82204; fTable_Si[580, 2] := 2.26608;
    fTable_Si[581, 0] := 1860; fTable_Si[581, 1] := 9.34866; fTable_Si[581, 2] := 4.09222;
    fTable_Si[582, 0] := 1890.08; fTable_Si[582, 1] := 10.4859; fTable_Si[582, 2] := 4.00184;
    fTable_Si[583, 0] := 1920.65; fTable_Si[583, 1] := 11.1017; fTable_Si[583, 2] := 3.91340;
    fTable_Si[584, 0] := 1951.72; fTable_Si[584, 1] := 11.5305; fTable_Si[584, 2] := 3.82687;
    fTable_Si[585, 0] := 1983.29; fTable_Si[585, 1] := 11.8609; fTable_Si[585, 2] := 3.74224;
    fTable_Si[586, 0] := 2015.37; fTable_Si[586, 1] := 12.1301; fTable_Si[586, 2] := 3.65896;
    fTable_Si[587, 0] := 2047.96; fTable_Si[587, 1] := 12.3571; fTable_Si[587, 2] := 3.57698;
    fTable_Si[588, 0] := 2081.09; fTable_Si[588, 1] := 12.5533; fTable_Si[588, 2] := 3.49664;
    fTable_Si[589, 0] := 2114.75; fTable_Si[589, 1] := 12.7254; fTable_Si[589, 2] := 3.41523;
    fTable_Si[590, 0] := 2148.95; fTable_Si[590, 1] := 12.8775; fTable_Si[590, 2] := 3.33521;
    fTable_Si[591, 0] := 2183.71; fTable_Si[591, 1] := 13.0131; fTable_Si[591, 2] := 3.25641;
    fTable_Si[592, 0] := 2219.03; fTable_Si[592, 1] := 13.1350; fTable_Si[592, 2] := 3.17868;
    fTable_Si[593, 0] := 2254.92; fTable_Si[593, 1] := 13.2452; fTable_Si[593, 2] := 3.10245;
    fTable_Si[594, 0] := 2291.39; fTable_Si[594, 1] := 13.3453; fTable_Si[594, 2] := 3.02741;
    fTable_Si[595, 0] := 2328.45; fTable_Si[595, 1] := 13.4369; fTable_Si[595, 2] := 2.95359;
    fTable_Si[596, 0] := 2366.11; fTable_Si[596, 1] := 13.5205; fTable_Si[596, 2] := 2.88121;
    fTable_Si[597, 0] := 2404.38; fTable_Si[597, 1] := 13.5972; fTable_Si[597, 2] := 2.80993;
    fTable_Si[598, 0] := 2443.27; fTable_Si[598, 1] := 13.6676; fTable_Si[598, 2] := 2.74011;
    fTable_Si[599, 0] := 2482.79; fTable_Si[599, 1] := 13.7324; fTable_Si[599, 2] := 2.67152;
    fTable_Si[600, 0] := 2522.95; fTable_Si[600, 1] := 13.7921; fTable_Si[600, 2] := 2.60424;
    fTable_Si[601, 0] := 2563.75; fTable_Si[601, 1] := 13.8472; fTable_Si[601, 2] := 2.53844;
    fTable_Si[602, 0] := 2605.22; fTable_Si[602, 1] := 13.8981; fTable_Si[602, 2] := 2.47374;
    fTable_Si[603, 0] := 2647.36; fTable_Si[603, 1] := 13.9449; fTable_Si[603, 2] := 2.41045;
    fTable_Si[604, 0] := 2690.18; fTable_Si[604, 1] := 13.9882; fTable_Si[604, 2] := 2.34854;
    fTable_Si[605, 0] := 2733.69; fTable_Si[605, 1] := 14.0282; fTable_Si[605, 2] := 2.28769;
    fTable_Si[606, 0] := 2777.90; fTable_Si[606, 1] := 14.0651; fTable_Si[606, 2] := 2.22827;
    fTable_Si[607, 0] := 2822.83; fTable_Si[607, 1] := 14.0991; fTable_Si[607, 2] := 2.17014;
    fTable_Si[608, 0] := 2868.49; fTable_Si[608, 1] := 14.1305; fTable_Si[608, 2] := 2.11320;
    fTable_Si[609, 0] := 2914.89; fTable_Si[609, 1] := 14.1594; fTable_Si[609, 2] := 2.05756;
    fTable_Si[610, 0] := 2962.03; fTable_Si[610, 1] := 14.1859; fTable_Si[610, 2] := 2.00307;
    fTable_Si[611, 0] := 3009.94; fTable_Si[611, 1] := 14.2104; fTable_Si[611, 2] := 1.94988;
    fTable_Si[612, 0] := 3058.62; fTable_Si[612, 1] := 14.2329; fTable_Si[612, 2] := 1.89788;
    fTable_Si[613, 0] := 3108.09; fTable_Si[613, 1] := 14.2535; fTable_Si[613, 2] := 1.84703;
    fTable_Si[614, 0] := 3158.37; fTable_Si[614, 1] := 14.2723; fTable_Si[614, 2] := 1.79742;
    fTable_Si[615, 0] := 3209.45; fTable_Si[615, 1] := 14.2894; fTable_Si[615, 2] := 1.74890;
    fTable_Si[616, 0] := 3261.36; fTable_Si[616, 1] := 14.3051; fTable_Si[616, 2] := 1.70154;
    fTable_Si[617, 0] := 3314.11; fTable_Si[617, 1] := 14.3194; fTable_Si[617, 2] := 1.65534;
    fTable_Si[618, 0] := 3367.71; fTable_Si[618, 1] := 14.3322; fTable_Si[618, 2] := 1.61015;
    fTable_Si[619, 0] := 3422.18; fTable_Si[619, 1] := 14.3438; fTable_Si[619, 2] := 1.56612;
    fTable_Si[620, 0] := 3477.53; fTable_Si[620, 1] := 14.3542; fTable_Si[620, 2] := 1.52314;
    fTable_Si[621, 0] := 3533.78; fTable_Si[621, 1] := 14.3635; fTable_Si[621, 2] := 1.48119;
    fTable_Si[622, 0] := 3590.94; fTable_Si[622, 1] := 14.3718; fTable_Si[622, 2] := 1.44032;
    fTable_Si[623, 0] := 3649.02; fTable_Si[623, 1] := 14.3791; fTable_Si[623, 2] := 1.40039;
    fTable_Si[624, 0] := 3708.04; fTable_Si[624, 1] := 14.3855; fTable_Si[624, 2] := 1.36149;
    fTable_Si[625, 0] := 3768.01; fTable_Si[625, 1] := 14.3910; fTable_Si[625, 2] := 1.32359;
    fTable_Si[626, 0] := 3828.96; fTable_Si[626, 1] := 14.3957; fTable_Si[626, 2] := 1.28658;
    fTable_Si[627, 0] := 3890.89; fTable_Si[627, 1] := 14.3997; fTable_Si[627, 2] := 1.25056;
    fTable_Si[628, 0] := 3953.82; fTable_Si[628, 1] := 14.4029; fTable_Si[628, 2] := 1.21543;
    fTable_Si[629, 0] := 4017.77; fTable_Si[629, 1] := 14.4055; fTable_Si[629, 2] := 1.18120;
    fTable_Si[630, 0] := 4082.75; fTable_Si[630, 1] := 14.4075; fTable_Si[630, 2] := 1.14788;
    fTable_Si[631, 0] := 4148.79; fTable_Si[631, 1] := 14.4089; fTable_Si[631, 2] := 1.11537;
    fTable_Si[632, 0] := 4215.89; fTable_Si[632, 1] := 14.4097; fTable_Si[632, 2] := 1.08375;
    fTable_Si[633, 0] := 4284.08; fTable_Si[633, 1] := 14.4101; fTable_Si[633, 2] := 1.05295;
    fTable_Si[634, 0] := 4353.37; fTable_Si[634, 1] := 14.4100; fTable_Si[634, 2] := 1.02294;
    fTable_Si[635, 0] := 4423.78; fTable_Si[635, 1] := 14.4094; fTable_Si[635, 2] := 0.993744;
    fTable_Si[636, 0] := 4495.33; fTable_Si[636, 1] := 14.4085; fTable_Si[636, 2] := 0.965295;
    fTable_Si[637, 0] := 4568.04; fTable_Si[637, 1] := 14.4071; fTable_Si[637, 2] := 0.937606;
    fTable_Si[638, 0] := 4641.93; fTable_Si[638, 1] := 14.4054; fTable_Si[638, 2] := 0.910663;
    fTable_Si[639, 0] := 4717.01; fTable_Si[639, 1] := 14.4034; fTable_Si[639, 2] := 0.884415;
    fTable_Si[640, 0] := 4793.30; fTable_Si[640, 1] := 14.4011; fTable_Si[640, 2] := 0.858896;
    fTable_Si[641, 0] := 4870.83; fTable_Si[641, 1] := 14.3984; fTable_Si[641, 2] := 0.834074;
    fTable_Si[642, 0] := 4949.61; fTable_Si[642, 1] := 14.3956; fTable_Si[642, 2] := 0.809917;
    fTable_Si[643, 0] := 5029.67; fTable_Si[643, 1] := 14.3925; fTable_Si[643, 2] := 0.786429;
    fTable_Si[644, 0] := 5111.02; fTable_Si[644, 1] := 14.3891; fTable_Si[644, 2] := 0.763535;
    fTable_Si[645, 0] := 5193.68; fTable_Si[645, 1] := 14.3856; fTable_Si[645, 2] := 0.741289;
    fTable_Si[646, 0] := 5277.69; fTable_Si[646, 1] := 14.3818; fTable_Si[646, 2] := 0.719672;
    fTable_Si[647, 0] := 5363.05; fTable_Si[647, 1] := 14.3779; fTable_Si[647, 2] := 0.698635;
    fTable_Si[648, 0] := 5449.79; fTable_Si[648, 1] := 14.3739; fTable_Si[648, 2] := 0.678189;
    fTable_Si[649, 0] := 5537.94; fTable_Si[649, 1] := 14.3697; fTable_Si[649, 2] := 0.658294;
    fTable_Si[650, 0] := 5627.51; fTable_Si[650, 1] := 14.3654; fTable_Si[650, 2] := 0.638950;
    fTable_Si[651, 0] := 5718.53; fTable_Si[651, 1] := 14.3609; fTable_Si[651, 2] := 0.620147;
    fTable_Si[652, 0] := 5811.02; fTable_Si[652, 1] := 14.3564; fTable_Si[652, 2] := 0.601873;
    fTable_Si[653, 0] := 5905.01; fTable_Si[653, 1] := 14.3517; fTable_Si[653, 2] := 0.584116;
    fTable_Si[654, 0] := 6000.52; fTable_Si[654, 1] := 14.3470; fTable_Si[654, 2] := 0.566843;
    fTable_Si[655, 0] := 6097.57; fTable_Si[655, 1] := 14.3422; fTable_Si[655, 2] := 0.550055;
    fTable_Si[656, 0] := 6196.20; fTable_Si[656, 1] := 14.3374; fTable_Si[656, 2] := 0.533751;
    fTable_Si[657, 0] := 6296.42; fTable_Si[657, 1] := 14.3325; fTable_Si[657, 2] := 0.517913;
    fTable_Si[658, 0] := 6349; fTable_Si[658, 1] := 14.3300; fTable_Si[658, 2] := 0.509889;
    fTable_Si[659, 0] := 6432; fTable_Si[659, 1] := 14.3259; fTable_Si[659, 2] := 0.497536;
    fTable_Si[660, 0] := 6536.03; fTable_Si[660, 1] := 14.3209; fTable_Si[660, 2] := 0.482727;
    fTable_Si[661, 0] := 6641.75; fTable_Si[661, 1] := 14.3159; fTable_Si[661, 2] := 0.468336;
    fTable_Si[662, 0] := 6749.17; fTable_Si[662, 1] := 14.3109; fTable_Si[662, 2] := 0.454339;
    fTable_Si[663, 0] := 6858.33; fTable_Si[663, 1] := 14.3059; fTable_Si[663, 2] := 0.440746;
    fTable_Si[664, 0] := 6969.26; fTable_Si[664, 1] := 14.3008; fTable_Si[664, 2] := 0.427550;
    fTable_Si[665, 0] := 7081.98; fTable_Si[665, 1] := 14.2958; fTable_Si[665, 2] := 0.414725;
    fTable_Si[666, 0] := 7196.53; fTable_Si[666, 1] := 14.2907; fTable_Si[666, 2] := 0.402271;
    fTable_Si[667, 0] := 7312.93; fTable_Si[667, 1] := 14.2857; fTable_Si[667, 2] := 0.390179;
    fTable_Si[668, 0] := 7431.21; fTable_Si[668, 1] := 14.2806; fTable_Si[668, 2] := 0.378427;
    fTable_Si[669, 0] := 7551.40; fTable_Si[669, 1] := 14.2756; fTable_Si[669, 2] := 0.367020;
    fTable_Si[670, 0] := 7673.54; fTable_Si[670, 1] := 14.2706; fTable_Si[670, 2] := 0.355946;
    fTable_Si[671, 0] := 7797.65; fTable_Si[671, 1] := 14.2657; fTable_Si[671, 2] := 0.345189;
    fTable_Si[672, 0] := 7923.77; fTable_Si[672, 1] := 14.2607; fTable_Si[672, 2] := 0.334747;
    fTable_Si[673, 0] := 8051.94; fTable_Si[673, 1] := 14.2558; fTable_Si[673, 2] := 0.324605;
    fTable_Si[674, 0] := 8182.17; fTable_Si[674, 1] := 14.2510; fTable_Si[674, 2] := 0.314762;
    fTable_Si[675, 0] := 8314.51; fTable_Si[675, 1] := 14.2461; fTable_Si[675, 2] := 0.305207;
    fTable_Si[676, 0] := 8448.99; fTable_Si[676, 1] := 14.2414; fTable_Si[676, 2] := 0.295929;
    fTable_Si[677, 0] := 8585.64; fTable_Si[677, 1] := 14.2366; fTable_Si[677, 2] := 0.286926;
    fTable_Si[678, 0] := 8724.51; fTable_Si[678, 1] := 14.2319; fTable_Si[678, 2] := 0.278183;
    fTable_Si[679, 0] := 8865.62; fTable_Si[679, 1] := 14.2273; fTable_Si[679, 2] := 0.269697;
    fTable_Si[680, 0] := 9009.02; fTable_Si[680, 1] := 14.2227; fTable_Si[680, 2] := 0.261465;
    fTable_Si[681, 0] := 9154.73; fTable_Si[681, 1] := 14.2181; fTable_Si[681, 2] := 0.253469;
    fTable_Si[682, 0] := 9302.80; fTable_Si[682, 1] := 14.2136; fTable_Si[682, 2] := 0.245713;
    fTable_Si[683, 0] := 9453.27; fTable_Si[683, 1] := 14.2091; fTable_Si[683, 2] := 0.238188;
    fTable_Si[684, 0] := 9606.17; fTable_Si[684, 1] := 14.2047; fTable_Si[684, 2] := 0.230880;
    fTable_Si[685, 0] := 9761.54; fTable_Si[685, 1] := 14.2004; fTable_Si[685, 2] := 0.223790;
    fTable_Si[686, 0] := 9919.42; fTable_Si[686, 1] := 14.1961; fTable_Si[686, 2] := 0.216911;
    fTable_Si[687, 0] := 10079.9; fTable_Si[687, 1] := 14.1919; fTable_Si[687, 2] := 0.210235;
    fTable_Si[688, 0] := 10242.9; fTable_Si[688, 1] := 14.1877; fTable_Si[688, 2] := 0.203758;
    fTable_Si[689, 0] := 10408.6; fTable_Si[689, 1] := 14.1836; fTable_Si[689, 2] := 0.197474;
    fTable_Si[690, 0] := 10576.9; fTable_Si[690, 1] := 14.1795; fTable_Si[690, 2] := 0.191376;
    fTable_Si[691, 0] := 10748.0; fTable_Si[691, 1] := 14.1756; fTable_Si[691, 2] := 0.185461;
    fTable_Si[692, 0] := 10921.8; fTable_Si[692, 1] := 14.1716; fTable_Si[692, 2] := 0.179721;
    fTable_Si[693, 0] := 11098.5; fTable_Si[693, 1] := 14.1677; fTable_Si[693, 2] := 0.174154;
    fTable_Si[694, 0] := 11278.0; fTable_Si[694, 1] := 14.1639; fTable_Si[694, 2] := 0.168752;
    fTable_Si[695, 0] := 11460.4; fTable_Si[695, 1] := 14.1602; fTable_Si[695, 2] := 0.163513;
    fTable_Si[696, 0] := 11645.8; fTable_Si[696, 1] := 14.1565; fTable_Si[696, 2] := 0.158430;
    fTable_Si[697, 0] := 11834.1; fTable_Si[697, 1] := 14.1528; fTable_Si[697, 2] := 0.153500;
    fTable_Si[698, 0] := 12025.5; fTable_Si[698, 1] := 14.1492; fTable_Si[698, 2] := 0.148717;
    fTable_Si[699, 0] := 12220.0; fTable_Si[699, 1] := 14.1457; fTable_Si[699, 2] := 0.144079;
    fTable_Si[700, 0] := 12417.7; fTable_Si[700, 1] := 14.1423; fTable_Si[700, 2] := 0.139580;
    fTable_Si[701, 0] := 12618.5; fTable_Si[701, 1] := 14.1389; fTable_Si[701, 2] := 0.135216;
    fTable_Si[702, 0] := 12822.6; fTable_Si[702, 1] := 14.1355; fTable_Si[702, 2] := 0.130984;
    fTable_Si[703, 0] := 13030.0; fTable_Si[703, 1] := 14.1322; fTable_Si[703, 2] := 0.126879;
    fTable_Si[704, 0] := 13240.8; fTable_Si[704, 1] := 14.1290; fTable_Si[704, 2] := 0.122899;
    fTable_Si[705, 0] := 13454.9; fTable_Si[705, 1] := 14.1258; fTable_Si[705, 2] := 0.119038;
    fTable_Si[706, 0] := 13672.6; fTable_Si[706, 1] := 14.1227; fTable_Si[706, 2] := 0.115294;
    fTable_Si[707, 0] := 13893.7; fTable_Si[707, 1] := 14.1197; fTable_Si[707, 2] := 0.111664;
    fTable_Si[708, 0] := 14118.4; fTable_Si[708, 1] := 14.1167; fTable_Si[708, 2] := 0.108143;
    fTable_Si[709, 0] := 14346.8; fTable_Si[709, 1] := 14.1137; fTable_Si[709, 2] := 0.104730;
    fTable_Si[710, 0] := 14578.8; fTable_Si[710, 1] := 14.1108; fTable_Si[710, 2] := 0.101419;
    fTable_Si[711, 0] := 14814.6; fTable_Si[711, 1] := 14.1080; fTable_Si[711, 2] := 0.0982093;
    fTable_Si[712, 0] := 15054.2; fTable_Si[712, 1] := 14.1052; fTable_Si[712, 2] := 0.0950968;
    fTable_Si[713, 0] := 15297.7; fTable_Si[713, 1] := 14.1025; fTable_Si[713, 2] := 0.0920790;
    fTable_Si[714, 0] := 15545.2; fTable_Si[714, 1] := 14.0998; fTable_Si[714, 2] := 0.0891530;
    fTable_Si[715, 0] := 15796.6; fTable_Si[715, 1] := 14.0972; fTable_Si[715, 2] := 0.0863160;
    fTable_Si[716, 0] := 16052.1; fTable_Si[716, 1] := 14.0946; fTable_Si[716, 2] := 0.0835654;
    fTable_Si[717, 0] := 16311.7; fTable_Si[717, 1] := 14.0921; fTable_Si[717, 2] := 0.0808987;
    fTable_Si[718, 0] := 16575.5; fTable_Si[718, 1] := 14.0896; fTable_Si[718, 2] := 0.0783132;
    fTable_Si[719, 0] := 16843.6; fTable_Si[719, 1] := 14.0872; fTable_Si[719, 2] := 0.0758067;
    fTable_Si[720, 0] := 17116.1; fTable_Si[720, 1] := 14.0848; fTable_Si[720, 2] := 0.0733767;
    fTable_Si[721, 0] := 17392.9; fTable_Si[721, 1] := 14.0825; fTable_Si[721, 2] := 0.0710210;
    fTable_Si[722, 0] := 17674.2; fTable_Si[722, 1] := 14.0802; fTable_Si[722, 2] := 0.0687373;
    fTable_Si[723, 0] := 17960.1; fTable_Si[723, 1] := 14.0780; fTable_Si[723, 2] := 0.0665234;
    fTable_Si[724, 0] := 18250.6; fTable_Si[724, 1] := 14.0758; fTable_Si[724, 2] := 0.0643773;
    fTable_Si[725, 0] := 18545.8; fTable_Si[725, 1] := 14.0736; fTable_Si[725, 2] := 0.0622970;
    fTable_Si[726, 0] := 18845.7; fTable_Si[726, 1] := 14.0715; fTable_Si[726, 2] := 0.0602804;
    fTable_Si[727, 0] := 19150.5; fTable_Si[727, 1] := 14.0695; fTable_Si[727, 2] := 0.0583256;
    fTable_Si[728, 0] := 19460.3; fTable_Si[728, 1] := 14.0675; fTable_Si[728, 2] := 0.0564308;
    fTable_Si[729, 0] := 19775.0; fTable_Si[729, 1] := 14.0655; fTable_Si[729, 2] := 0.0545942;
    fTable_Si[730, 0] := 20094.9; fTable_Si[730, 1] := 14.0636; fTable_Si[730, 2] := 0.0528124;
    fTable_Si[731, 0] := 20419.9; fTable_Si[731, 1] := 14.0617; fTable_Si[731, 2] := 0.0510884;
    fTable_Si[732, 0] := 20750.2; fTable_Si[732, 1] := 14.0598; fTable_Si[732, 2] := 0.0494193;
    fTable_Si[733, 0] := 21085.8; fTable_Si[733, 1] := 14.0580; fTable_Si[733, 2] := 0.0478034;
    fTable_Si[734, 0] := 21426.8; fTable_Si[734, 1] := 14.0562; fTable_Si[734, 2] := 0.0462390;
    fTable_Si[735, 0] := 21773.4; fTable_Si[735, 1] := 14.0545; fTable_Si[735, 2] := 0.0447245;
    fTable_Si[736, 0] := 22125.6; fTable_Si[736, 1] := 14.0528; fTable_Si[736, 2] := 0.0432583;
    fTable_Si[737, 0] := 22483.4; fTable_Si[737, 1] := 14.0511; fTable_Si[737, 2] := 0.0418390;
    fTable_Si[738, 0] := 22847.1; fTable_Si[738, 1] := 14.0495; fTable_Si[738, 2] := 0.0404650;
    fTable_Si[739, 0] := 23216.6; fTable_Si[739, 1] := 14.0479; fTable_Si[739, 2] := 0.0391349;
    fTable_Si[740, 0] := 23592.1; fTable_Si[740, 1] := 14.0463; fTable_Si[740, 2] := 0.0378475;
    fTable_Si[741, 0] := 23973.7; fTable_Si[741, 1] := 14.0448; fTable_Si[741, 2] := 0.0366013;
    fTable_Si[742, 0] := 24361.5; fTable_Si[742, 1] := 14.0433; fTable_Si[742, 2] := 0.0353950;
    fTable_Si[743, 0] := 24755.5; fTable_Si[743, 1] := 14.0419; fTable_Si[743, 2] := 0.0342274;
    fTable_Si[744, 0] := 25155.9; fTable_Si[744, 1] := 14.0405; fTable_Si[744, 2] := 0.0330973;
    fTable_Si[745, 0] := 25562.8; fTable_Si[745, 1] := 14.0391; fTable_Si[745, 2] := 0.0320035;
    fTable_Si[746, 0] := 25976.2; fTable_Si[746, 1] := 14.0377; fTable_Si[746, 2] := 0.0309448;
    fTable_Si[747, 0] := 26396.4; fTable_Si[747, 1] := 14.0364; fTable_Si[747, 2] := 0.0299202;
    fTable_Si[748, 0] := 26823.3; fTable_Si[748, 1] := 14.0351; fTable_Si[748, 2] := 0.0289286;
    fTable_Si[749, 0] := 27257.2; fTable_Si[749, 1] := 14.0338; fTable_Si[749, 2] := 0.0279690;
    fTable_Si[750, 0] := 27698.0; fTable_Si[750, 1] := 14.0326; fTable_Si[750, 2] := 0.0270403;
    fTable_Si[751, 0] := 28146.0; fTable_Si[751, 1] := 14.0314; fTable_Si[751, 2] := 0.0261415;
    fTable_Si[752, 0] := 28601.3; fTable_Si[752, 1] := 14.0302; fTable_Si[752, 2] := 0.0252718;
    fTable_Si[753, 0] := 29063.9; fTable_Si[753, 1] := 14.0291; fTable_Si[753, 2] := 0.0244301;
    fTable_Si[754, 0] := 29533.9; fTable_Si[754, 1] := 14.0279; fTable_Si[754, 2] := 0.0236157;
    fTable_Si[755, 0] := 30000.0; fTable_Si[755, 1] := 14.0269; fTable_Si[755, 2] := 0.0228464;

    bInit := TRUE;
END_IF

(* Get correct table *)


IF sTableName = 'Ge' THEN
    iRowSize := ADR(fTable_Ge[1,0]) - ADR(fTable_Ge[0,0]);
    iRowCount := 505;
    fRow1 := ADR(fTable_Ge[0, 0]);
    fTableLookupLow := 10.0000;
    fTableLookupHigh := 30000.0;
ELSIF sTableName = 'C' OR sTableName = 'C (Diamond)' THEN
    iRowSize := ADR(fTable_C[1,0]) - ADR(fTable_C[0,0]);
    iRowCount := 501;
    fRow1 := ADR(fTable_C[0, 0]);
    fTableLookupLow := 10.0000;
    fTableLookupHigh := 30000.0;
ELSIF sTableName = 'Al' THEN
    iRowSize := ADR(fTable_Al[1,0]) - ADR(fTable_Al[0,0]);
    iRowCount := 503;
    fRow1 := ADR(fTable_Al[0, 0]);
    fTableLookupLow := 10.0000;
    fTableLookupHigh := 30000.0;
ELSIF sTableName = 'Be' THEN
    iRowSize := ADR(fTable_Be[1,0]) - ADR(fTable_Be[0,0]);
    iRowCount := 723;
    fRow1 := ADR(fTable_Be[0, 0]);
    fTableLookupLow := 10.0000;
    fTableLookupHigh := 30000.0;
ELSIF sTableName = 'Si' THEN
    iRowSize := ADR(fTable_Si[1,0]) - ADR(fTable_Si[0,0]);
    iRowCount := 755;
    fRow1 := ADR(fTable_Si[0, 0]);
    fTableLookupLow := 10.0000;
    fTableLookupHigh := 30000.0;
ELSE
    bError := TRUE;
    bDone := TRUE;
    RETURN;
END_IF

IF fEnergyEV < fTableLookupLow THEN
    bDone := TRUE;
    RETURN;
ELSIF fEnergyEV > fTableLookupHigh THEN
    bDone := TRUE;
    RETURN;
END_IF

FOR iRowIdx := 0 TO iRowCount - 1
DO
    fRow2 := fRow1 + iRowSize;
    IF fEnergyEV >= fRow1^[0] AND fEnergyEV <= fRow2^[0] THEN
        fEnergyEV_RowDelta := fRow2^[0] - fRow1^[0];
        IF fEnergyEV_RowDelta <= 0.0 THEN
            bFound := TRUE;
            bError := TRUE;
            bDone := TRUE;
        ELSE

            // Interpolate output: f1
            fSlope := (fRow2^[1] - fRow1^[1]) / fEnergyEV_RowDelta;
            f1 := fRow1^[1] + fSlope * (fEnergyEV - fRow1^[0]);

            // Interpolate output: f2
            fSlope := (fRow2^[2] - fRow1^[2]) / fEnergyEV_RowDelta;
            f2 := fRow1^[2] + fSlope * (fEnergyEV - fRow1^[0]);

            bFound := TRUE;
            bError := FALSE;
            bDone := TRUE;
        END_IF
        RETURN;
    END_IF
    fRow1 := fRow2;
END_FOR

END_FUNCTION_BLOCK

(* stored: Version 1.1.0.1
   POU FB_ScatteringFactorLUT: Id {01ad8d01-6b90-c34c-086b-4fed4a9c1079}, SpecialFunc None *)
